// TwinCAT 3 PLC project lcls_plc_dream_vac
// ProgramVersion: 3.1.4022.7
// libraries:
//   LCLS General, * (SLAC)
//   LCLS Vacuum, * (SLAC - LCLS)
//   LCLSVacuumSerialDriverLib, * (SLAC - LCLS)
//   PMPS, * (SLAC - LCLS)
//   Tc2_SerialCom, * (Beckhoff Automation GmbH)
//   Tc2_Standard, * (Beckhoff Automation GmbH)
//   Tc2_System, * (Beckhoff Automation GmbH)
//   Tc2_Utilities, * (Beckhoff Automation GmbH)
//   Tc3_Module, * (Beckhoff Automation GmbH)
// project tree:
//   DUTs/ ST_TD400Control.TcDUT (not stored), ST_TD400Status.TcDUT (not stored)
//   GVLs/ GVL_FWM.TcGVL (not stored), GVL_PLC_Interface.TcGVL (not stored), GVL_Serial_Com.TcGVL (not stored), GVL_VAC_GAUGES.TcGVL (not stored), GVL_VAC_PUMPS.TcGVL (not stored), GVL_VAC_VALVES.TcGVL (not stored), GVL_Variables.TcGVL (not stored)
//   / PlcTask.TcTTO (not stored), Serial_COM.TcTTO (not stored)
//   POUs/Functions/ F_TurboIlkLogic.TcPOU (not stored)
//   POUs/ MAIN.TcPOU (not stored), PRG_COM.TcPOU (not stored), PRG_ECAT_CHECK.TcPOU (not stored), PRG_GAUGES.TcPOU (not stored), PRG_HV_ILK.TcPOU (not stored), PRG_COIL_PS_ILK.TcPOU (not stored), PRG_TURBO_PUMPS.TcPOU (not stored), PRG_VALVES.TcPOU (not stored)
//   POUs/TD400_Test/ FB_OERLIKON_TD400_COM.TcPOU, FB_OERLIKON_TD400_TO_PTM.TcPOU, FB_TD400SerialDriver.TcPOU (not stored), FB_TD400Transaction.TcPOU (not stored), F_CalcTD400Checksum.TcPOU (not stored)
//   POUs/TempFB_IE514/ FB_IE514.TcPOU (not stored)
// real-time tasks:
//   TASK PlcTask: cycle T#10ms, priority 20, ADS port 350
//   TASK Serial_COM: cycle T#2ms, priority 19, ADS port 351
// I/O:
//   DEVICE Device 1 (EtherCAT)
// variable links:
//   lcls_plc_dream_vac Instance <-> Device 1 (EtherCAT)/R20_DRL_03_CX0_EK1200/R20_DRL_03_E10_EL6001
//     Serial_COM Inputs/GVL_Serial_Com.stComIn_DREAM_DP3_PTM_01/D[0] <-> COM Inputs/Data In 0
//     Serial_COM Inputs/GVL_Serial_Com.stComIn_DREAM_DP3_PTM_01/D[10] <-> COM Inputs/Data In 10
//     Serial_COM Inputs/GVL_Serial_Com.stComIn_DREAM_DP3_PTM_01/D[11] <-> COM Inputs/Data In 11
//     Serial_COM Inputs/GVL_Serial_Com.stComIn_DREAM_DP3_PTM_01/D[12] <-> COM Inputs/Data In 12
//     Serial_COM Inputs/GVL_Serial_Com.stComIn_DREAM_DP3_PTM_01/D[13] <-> COM Inputs/Data In 13
//     Serial_COM Inputs/GVL_Serial_Com.stComIn_DREAM_DP3_PTM_01/D[14] <-> COM Inputs/Data In 14
//     Serial_COM Inputs/GVL_Serial_Com.stComIn_DREAM_DP3_PTM_01/D[15] <-> COM Inputs/Data In 15
//     Serial_COM Inputs/GVL_Serial_Com.stComIn_DREAM_DP3_PTM_01/D[16] <-> COM Inputs/Data In 16
//     Serial_COM Inputs/GVL_Serial_Com.stComIn_DREAM_DP3_PTM_01/D[17] <-> COM Inputs/Data In 17
//     Serial_COM Inputs/GVL_Serial_Com.stComIn_DREAM_DP3_PTM_01/D[18] <-> COM Inputs/Data In 18
//     Serial_COM Inputs/GVL_Serial_Com.stComIn_DREAM_DP3_PTM_01/D[19] <-> COM Inputs/Data In 19
//     Serial_COM Inputs/GVL_Serial_Com.stComIn_DREAM_DP3_PTM_01/D[1] <-> COM Inputs/Data In 1
//     Serial_COM Inputs/GVL_Serial_Com.stComIn_DREAM_DP3_PTM_01/D[20] <-> COM Inputs/Data In 20
//     Serial_COM Inputs/GVL_Serial_Com.stComIn_DREAM_DP3_PTM_01/D[21] <-> COM Inputs/Data In 21
//     Serial_COM Inputs/GVL_Serial_Com.stComIn_DREAM_DP3_PTM_01/D[2] <-> COM Inputs/Data In 2
//     Serial_COM Inputs/GVL_Serial_Com.stComIn_DREAM_DP3_PTM_01/D[3] <-> COM Inputs/Data In 3
//     Serial_COM Inputs/GVL_Serial_Com.stComIn_DREAM_DP3_PTM_01/D[4] <-> COM Inputs/Data In 4
//     Serial_COM Inputs/GVL_Serial_Com.stComIn_DREAM_DP3_PTM_01/D[5] <-> COM Inputs/Data In 5
//     Serial_COM Inputs/GVL_Serial_Com.stComIn_DREAM_DP3_PTM_01/D[6] <-> COM Inputs/Data In 6
//     Serial_COM Inputs/GVL_Serial_Com.stComIn_DREAM_DP3_PTM_01/D[7] <-> COM Inputs/Data In 7
//     Serial_COM Inputs/GVL_Serial_Com.stComIn_DREAM_DP3_PTM_01/D[8] <-> COM Inputs/Data In 8
//     Serial_COM Inputs/GVL_Serial_Com.stComIn_DREAM_DP3_PTM_01/D[9] <-> COM Inputs/Data In 9
//     Serial_COM Inputs/GVL_Serial_Com.stComIn_DREAM_DP3_PTM_01/Status <-> COM Inputs/Status
//     Serial_COM Outputs/GVL_Serial_Com.stComOut_DREAM_DP3_PTM_01/Ctrl <-> COM Outputs/Ctrl
//     Serial_COM Outputs/GVL_Serial_Com.stComOut_DREAM_DP3_PTM_01/D[0] <-> COM Outputs/Data Out 0
//     Serial_COM Outputs/GVL_Serial_Com.stComOut_DREAM_DP3_PTM_01/D[10] <-> COM Outputs/Data Out 10
//     Serial_COM Outputs/GVL_Serial_Com.stComOut_DREAM_DP3_PTM_01/D[11] <-> COM Outputs/Data Out 11
//     Serial_COM Outputs/GVL_Serial_Com.stComOut_DREAM_DP3_PTM_01/D[12] <-> COM Outputs/Data Out 12
//     Serial_COM Outputs/GVL_Serial_Com.stComOut_DREAM_DP3_PTM_01/D[13] <-> COM Outputs/Data Out 13
//     Serial_COM Outputs/GVL_Serial_Com.stComOut_DREAM_DP3_PTM_01/D[14] <-> COM Outputs/Data Out 14
//     Serial_COM Outputs/GVL_Serial_Com.stComOut_DREAM_DP3_PTM_01/D[15] <-> COM Outputs/Data Out 15
//     Serial_COM Outputs/GVL_Serial_Com.stComOut_DREAM_DP3_PTM_01/D[16] <-> COM Outputs/Data Out 16
//     Serial_COM Outputs/GVL_Serial_Com.stComOut_DREAM_DP3_PTM_01/D[17] <-> COM Outputs/Data Out 17
//     Serial_COM Outputs/GVL_Serial_Com.stComOut_DREAM_DP3_PTM_01/D[18] <-> COM Outputs/Data Out 18
//     Serial_COM Outputs/GVL_Serial_Com.stComOut_DREAM_DP3_PTM_01/D[19] <-> COM Outputs/Data Out 19
//     Serial_COM Outputs/GVL_Serial_Com.stComOut_DREAM_DP3_PTM_01/D[1] <-> COM Outputs/Data Out 1
//     Serial_COM Outputs/GVL_Serial_Com.stComOut_DREAM_DP3_PTM_01/D[20] <-> COM Outputs/Data Out 20
//     Serial_COM Outputs/GVL_Serial_Com.stComOut_DREAM_DP3_PTM_01/D[21] <-> COM Outputs/Data Out 21
//     Serial_COM Outputs/GVL_Serial_Com.stComOut_DREAM_DP3_PTM_01/D[2] <-> COM Outputs/Data Out 2
//     Serial_COM Outputs/GVL_Serial_Com.stComOut_DREAM_DP3_PTM_01/D[3] <-> COM Outputs/Data Out 3
//     Serial_COM Outputs/GVL_Serial_Com.stComOut_DREAM_DP3_PTM_01/D[4] <-> COM Outputs/Data Out 4
//     Serial_COM Outputs/GVL_Serial_Com.stComOut_DREAM_DP3_PTM_01/D[5] <-> COM Outputs/Data Out 5
//     Serial_COM Outputs/GVL_Serial_Com.stComOut_DREAM_DP3_PTM_01/D[6] <-> COM Outputs/Data Out 6
//     Serial_COM Outputs/GVL_Serial_Com.stComOut_DREAM_DP3_PTM_01/D[7] <-> COM Outputs/Data Out 7
//     Serial_COM Outputs/GVL_Serial_Com.stComOut_DREAM_DP3_PTM_01/D[8] <-> COM Outputs/Data Out 8
//     Serial_COM Outputs/GVL_Serial_Com.stComOut_DREAM_DP3_PTM_01/D[9] <-> COM Outputs/Data Out 9
//   lcls_plc_dream_vac Instance <-> Device 1 (EtherCAT)/R20_DRL_03_CX0_EK1200/R20_DRL_03_E11_EL6001
//     Serial_COM Inputs/GVL_Serial_Com.stComIn_DREAM_MC_PTM_01/D[0] <-> COM Inputs/Data In 0
//     Serial_COM Inputs/GVL_Serial_Com.stComIn_DREAM_MC_PTM_01/D[10] <-> COM Inputs/Data In 10
//     Serial_COM Inputs/GVL_Serial_Com.stComIn_DREAM_MC_PTM_01/D[11] <-> COM Inputs/Data In 11
//     Serial_COM Inputs/GVL_Serial_Com.stComIn_DREAM_MC_PTM_01/D[12] <-> COM Inputs/Data In 12
//     Serial_COM Inputs/GVL_Serial_Com.stComIn_DREAM_MC_PTM_01/D[13] <-> COM Inputs/Data In 13
//     Serial_COM Inputs/GVL_Serial_Com.stComIn_DREAM_MC_PTM_01/D[14] <-> COM Inputs/Data In 14
//     Serial_COM Inputs/GVL_Serial_Com.stComIn_DREAM_MC_PTM_01/D[15] <-> COM Inputs/Data In 15
//     Serial_COM Inputs/GVL_Serial_Com.stComIn_DREAM_MC_PTM_01/D[16] <-> COM Inputs/Data In 16
//     Serial_COM Inputs/GVL_Serial_Com.stComIn_DREAM_MC_PTM_01/D[17] <-> COM Inputs/Data In 17
//     Serial_COM Inputs/GVL_Serial_Com.stComIn_DREAM_MC_PTM_01/D[18] <-> COM Inputs/Data In 18
//     Serial_COM Inputs/GVL_Serial_Com.stComIn_DREAM_MC_PTM_01/D[19] <-> COM Inputs/Data In 19
//     Serial_COM Inputs/GVL_Serial_Com.stComIn_DREAM_MC_PTM_01/D[1] <-> COM Inputs/Data In 1
//     Serial_COM Inputs/GVL_Serial_Com.stComIn_DREAM_MC_PTM_01/D[20] <-> COM Inputs/Data In 20
//     Serial_COM Inputs/GVL_Serial_Com.stComIn_DREAM_MC_PTM_01/D[21] <-> COM Inputs/Data In 21
//     Serial_COM Inputs/GVL_Serial_Com.stComIn_DREAM_MC_PTM_01/D[2] <-> COM Inputs/Data In 2
//     Serial_COM Inputs/GVL_Serial_Com.stComIn_DREAM_MC_PTM_01/D[3] <-> COM Inputs/Data In 3
//     Serial_COM Inputs/GVL_Serial_Com.stComIn_DREAM_MC_PTM_01/D[4] <-> COM Inputs/Data In 4
//     Serial_COM Inputs/GVL_Serial_Com.stComIn_DREAM_MC_PTM_01/D[5] <-> COM Inputs/Data In 5
//     Serial_COM Inputs/GVL_Serial_Com.stComIn_DREAM_MC_PTM_01/D[6] <-> COM Inputs/Data In 6
//     Serial_COM Inputs/GVL_Serial_Com.stComIn_DREAM_MC_PTM_01/D[7] <-> COM Inputs/Data In 7
//     Serial_COM Inputs/GVL_Serial_Com.stComIn_DREAM_MC_PTM_01/D[8] <-> COM Inputs/Data In 8
//     Serial_COM Inputs/GVL_Serial_Com.stComIn_DREAM_MC_PTM_01/D[9] <-> COM Inputs/Data In 9
//     Serial_COM Inputs/GVL_Serial_Com.stComIn_DREAM_MC_PTM_01/Status <-> COM Inputs/Status
//     Serial_COM Outputs/GVL_Serial_Com.stComOut_DREAM_MC_PTM_01/Ctrl <-> COM Outputs/Ctrl
//     Serial_COM Outputs/GVL_Serial_Com.stComOut_DREAM_MC_PTM_01/D[0] <-> COM Outputs/Data Out 0
//     Serial_COM Outputs/GVL_Serial_Com.stComOut_DREAM_MC_PTM_01/D[10] <-> COM Outputs/Data Out 10
//     Serial_COM Outputs/GVL_Serial_Com.stComOut_DREAM_MC_PTM_01/D[11] <-> COM Outputs/Data Out 11
//     Serial_COM Outputs/GVL_Serial_Com.stComOut_DREAM_MC_PTM_01/D[12] <-> COM Outputs/Data Out 12
//     Serial_COM Outputs/GVL_Serial_Com.stComOut_DREAM_MC_PTM_01/D[13] <-> COM Outputs/Data Out 13
//     Serial_COM Outputs/GVL_Serial_Com.stComOut_DREAM_MC_PTM_01/D[14] <-> COM Outputs/Data Out 14
//     Serial_COM Outputs/GVL_Serial_Com.stComOut_DREAM_MC_PTM_01/D[15] <-> COM Outputs/Data Out 15
//     Serial_COM Outputs/GVL_Serial_Com.stComOut_DREAM_MC_PTM_01/D[16] <-> COM Outputs/Data Out 16
//     Serial_COM Outputs/GVL_Serial_Com.stComOut_DREAM_MC_PTM_01/D[17] <-> COM Outputs/Data Out 17
//     Serial_COM Outputs/GVL_Serial_Com.stComOut_DREAM_MC_PTM_01/D[18] <-> COM Outputs/Data Out 18
//     Serial_COM Outputs/GVL_Serial_Com.stComOut_DREAM_MC_PTM_01/D[19] <-> COM Outputs/Data Out 19
//     Serial_COM Outputs/GVL_Serial_Com.stComOut_DREAM_MC_PTM_01/D[1] <-> COM Outputs/Data Out 1
//     Serial_COM Outputs/GVL_Serial_Com.stComOut_DREAM_MC_PTM_01/D[20] <-> COM Outputs/Data Out 20
//     Serial_COM Outputs/GVL_Serial_Com.stComOut_DREAM_MC_PTM_01/D[21] <-> COM Outputs/Data Out 21
//     Serial_COM Outputs/GVL_Serial_Com.stComOut_DREAM_MC_PTM_01/D[2] <-> COM Outputs/Data Out 2
//     Serial_COM Outputs/GVL_Serial_Com.stComOut_DREAM_MC_PTM_01/D[3] <-> COM Outputs/Data Out 3
//     Serial_COM Outputs/GVL_Serial_Com.stComOut_DREAM_MC_PTM_01/D[4] <-> COM Outputs/Data Out 4
//     Serial_COM Outputs/GVL_Serial_Com.stComOut_DREAM_MC_PTM_01/D[5] <-> COM Outputs/Data Out 5
//     Serial_COM Outputs/GVL_Serial_Com.stComOut_DREAM_MC_PTM_01/D[6] <-> COM Outputs/Data Out 6
//     Serial_COM Outputs/GVL_Serial_Com.stComOut_DREAM_MC_PTM_01/D[7] <-> COM Outputs/Data Out 7
//     Serial_COM Outputs/GVL_Serial_Com.stComOut_DREAM_MC_PTM_01/D[8] <-> COM Outputs/Data Out 8
//     Serial_COM Outputs/GVL_Serial_Com.stComOut_DREAM_MC_PTM_01/D[9] <-> COM Outputs/Data Out 9
//   lcls_plc_dream_vac Instance <-> Device 1 (EtherCAT)/R20_DRL_03_CX0_EK1200/R20_DRL_03_E12_EL6001
//     Serial_COM Inputs/GVL_Serial_Com.stComIn_DREAM_MC_PTM_02/D[0] <-> COM Inputs/Data In 0
//     Serial_COM Inputs/GVL_Serial_Com.stComIn_DREAM_MC_PTM_02/D[10] <-> COM Inputs/Data In 10
//     Serial_COM Inputs/GVL_Serial_Com.stComIn_DREAM_MC_PTM_02/D[11] <-> COM Inputs/Data In 11
//     Serial_COM Inputs/GVL_Serial_Com.stComIn_DREAM_MC_PTM_02/D[12] <-> COM Inputs/Data In 12
//     Serial_COM Inputs/GVL_Serial_Com.stComIn_DREAM_MC_PTM_02/D[13] <-> COM Inputs/Data In 13
//     Serial_COM Inputs/GVL_Serial_Com.stComIn_DREAM_MC_PTM_02/D[14] <-> COM Inputs/Data In 14
//     Serial_COM Inputs/GVL_Serial_Com.stComIn_DREAM_MC_PTM_02/D[15] <-> COM Inputs/Data In 15
//     Serial_COM Inputs/GVL_Serial_Com.stComIn_DREAM_MC_PTM_02/D[16] <-> COM Inputs/Data In 16
//     Serial_COM Inputs/GVL_Serial_Com.stComIn_DREAM_MC_PTM_02/D[17] <-> COM Inputs/Data In 17
//     Serial_COM Inputs/GVL_Serial_Com.stComIn_DREAM_MC_PTM_02/D[18] <-> COM Inputs/Data In 18
//     Serial_COM Inputs/GVL_Serial_Com.stComIn_DREAM_MC_PTM_02/D[19] <-> COM Inputs/Data In 19
//     Serial_COM Inputs/GVL_Serial_Com.stComIn_DREAM_MC_PTM_02/D[1] <-> COM Inputs/Data In 1
//     Serial_COM Inputs/GVL_Serial_Com.stComIn_DREAM_MC_PTM_02/D[20] <-> COM Inputs/Data In 20
//     Serial_COM Inputs/GVL_Serial_Com.stComIn_DREAM_MC_PTM_02/D[21] <-> COM Inputs/Data In 21
//     Serial_COM Inputs/GVL_Serial_Com.stComIn_DREAM_MC_PTM_02/D[2] <-> COM Inputs/Data In 2
//     Serial_COM Inputs/GVL_Serial_Com.stComIn_DREAM_MC_PTM_02/D[3] <-> COM Inputs/Data In 3
//     Serial_COM Inputs/GVL_Serial_Com.stComIn_DREAM_MC_PTM_02/D[4] <-> COM Inputs/Data In 4
//     Serial_COM Inputs/GVL_Serial_Com.stComIn_DREAM_MC_PTM_02/D[5] <-> COM Inputs/Data In 5
//     Serial_COM Inputs/GVL_Serial_Com.stComIn_DREAM_MC_PTM_02/D[6] <-> COM Inputs/Data In 6
//     Serial_COM Inputs/GVL_Serial_Com.stComIn_DREAM_MC_PTM_02/D[7] <-> COM Inputs/Data In 7
//     Serial_COM Inputs/GVL_Serial_Com.stComIn_DREAM_MC_PTM_02/D[8] <-> COM Inputs/Data In 8
//     Serial_COM Inputs/GVL_Serial_Com.stComIn_DREAM_MC_PTM_02/D[9] <-> COM Inputs/Data In 9
//     Serial_COM Inputs/GVL_Serial_Com.stComIn_DREAM_MC_PTM_02/Status <-> COM Inputs/Status
//     Serial_COM Outputs/GVL_Serial_Com.stComOut_DREAM_MC_PTM_02/Ctrl <-> COM Outputs/Ctrl
//     Serial_COM Outputs/GVL_Serial_Com.stComOut_DREAM_MC_PTM_02/D[0] <-> COM Outputs/Data Out 0
//     Serial_COM Outputs/GVL_Serial_Com.stComOut_DREAM_MC_PTM_02/D[10] <-> COM Outputs/Data Out 10
//     Serial_COM Outputs/GVL_Serial_Com.stComOut_DREAM_MC_PTM_02/D[11] <-> COM Outputs/Data Out 11
//     Serial_COM Outputs/GVL_Serial_Com.stComOut_DREAM_MC_PTM_02/D[12] <-> COM Outputs/Data Out 12
//     Serial_COM Outputs/GVL_Serial_Com.stComOut_DREAM_MC_PTM_02/D[13] <-> COM Outputs/Data Out 13
//     Serial_COM Outputs/GVL_Serial_Com.stComOut_DREAM_MC_PTM_02/D[14] <-> COM Outputs/Data Out 14
//     Serial_COM Outputs/GVL_Serial_Com.stComOut_DREAM_MC_PTM_02/D[15] <-> COM Outputs/Data Out 15
//     Serial_COM Outputs/GVL_Serial_Com.stComOut_DREAM_MC_PTM_02/D[16] <-> COM Outputs/Data Out 16
//     Serial_COM Outputs/GVL_Serial_Com.stComOut_DREAM_MC_PTM_02/D[17] <-> COM Outputs/Data Out 17
//     Serial_COM Outputs/GVL_Serial_Com.stComOut_DREAM_MC_PTM_02/D[18] <-> COM Outputs/Data Out 18
//     Serial_COM Outputs/GVL_Serial_Com.stComOut_DREAM_MC_PTM_02/D[19] <-> COM Outputs/Data Out 19
//     Serial_COM Outputs/GVL_Serial_Com.stComOut_DREAM_MC_PTM_02/D[1] <-> COM Outputs/Data Out 1
//     Serial_COM Outputs/GVL_Serial_Com.stComOut_DREAM_MC_PTM_02/D[20] <-> COM Outputs/Data Out 20
//     Serial_COM Outputs/GVL_Serial_Com.stComOut_DREAM_MC_PTM_02/D[21] <-> COM Outputs/Data Out 21
//     Serial_COM Outputs/GVL_Serial_Com.stComOut_DREAM_MC_PTM_02/D[2] <-> COM Outputs/Data Out 2
//     Serial_COM Outputs/GVL_Serial_Com.stComOut_DREAM_MC_PTM_02/D[3] <-> COM Outputs/Data Out 3
//     Serial_COM Outputs/GVL_Serial_Com.stComOut_DREAM_MC_PTM_02/D[4] <-> COM Outputs/Data Out 4
//     Serial_COM Outputs/GVL_Serial_Com.stComOut_DREAM_MC_PTM_02/D[5] <-> COM Outputs/Data Out 5
//     Serial_COM Outputs/GVL_Serial_Com.stComOut_DREAM_MC_PTM_02/D[6] <-> COM Outputs/Data Out 6
//     Serial_COM Outputs/GVL_Serial_Com.stComOut_DREAM_MC_PTM_02/D[7] <-> COM Outputs/Data Out 7
//     Serial_COM Outputs/GVL_Serial_Com.stComOut_DREAM_MC_PTM_02/D[8] <-> COM Outputs/Data Out 8
//     Serial_COM Outputs/GVL_Serial_Com.stComOut_DREAM_MC_PTM_02/D[9] <-> COM Outputs/Data Out 9
//   lcls_plc_dream_vac Instance <-> Device 1 (EtherCAT)/R20_DRL_03_CX0_EK1200/R20_DRL_03_E14_EL6695
//     PlcTask Inputs/GVL_PLC_Interface.bEcatBridge_External_device_not_connected <-> SYNC Inputs/External device not connected
//     PlcTask Inputs/GVL_PLC_Interface.bEcatBridge_TxPDO_state <-> SYNC Inputs/TxPDO state
//     PlcTask Inputs/GVL_PLC_Interface.bEcatBridge_WcState <-> WcState/WcStateIn
//     PlcTask Inputs/GVL_PLC_Interface.sHUTCH_PLC_NAME <-> IO Inputs/HUTCH_PLC_NAME
//     PlcTask Outputs/GVL_PLC_Interface.bDREAM_HV_SAFETY_ENABLE <-> IO Outputs/DREAM_HV_SAFETY_ENABLE
//     PlcTask Outputs/GVL_PLC_Interface.bDREAM_MAIN_xAT_VAC <-> IO Outputs/DREAM_MAIN_xAT_VAC
//     PlcTask Outputs/GVL_PLC_Interface.bDREAM_MAIN_xPRESS_OK <-> IO Outputs/DREAM_MAIN_xPRESS_OK
//     PlcTask Outputs/GVL_PLC_Interface.bDREAM_TURBOS_ALL_AtSpd <-> IO Outputs/DREAM_TURBOS_ALL_AtSpd
//     PlcTask Outputs/GVL_PLC_Interface.fDREAM_MAIN_rPRESS <-> IO Outputs/DREAM_MAIN_rPRESS
//     PlcTask Outputs/GVL_PLC_Interface.sENDSTATION_PLC_NAME <-> IO Outputs/ENDSTATION_PLC_NAME
//   lcls_plc_dream_vac Instance <-> Device 1 (EtherCAT)/R20_DRL_03_CX0_EK1200/R20_DRL_03_E15_EL1122/K4S8_DRL_03_EK0_EK1100/K4S8_DRL_03_E10_EL1004
//     PlcTask Inputs/GVL_VAC_VALVES.DREAM_DP1_VRC_01.i_xClsLS <-> Channel 2/Input
//     PlcTask Inputs/GVL_VAC_VALVES.DREAM_DP1_VRC_02.i_xClsLS <-> Channel 4/Input
//     PlcTask Inputs/GVL_VAC_VALVES.DREAM_DP1_VRC_01.i_xOpnLS <-> Channel 1/Input
//     PlcTask Inputs/GVL_VAC_VALVES.DREAM_DP1_VRC_02.i_xOpnLS <-> Channel 3/Input
//   lcls_plc_dream_vac Instance <-> Device 1 (EtherCAT)/R20_DRL_03_CX0_EK1200/R20_DRL_03_E15_EL1122/K4S8_DRL_03_EK0_EK1100/K4S8_DRL_03_E11_EL2004
//     PlcTask Outputs/GVL_VAC_VALVES.DREAM_DP1_VRC_01.q_xOPN_DO <-> Channel 2/Output
//     PlcTask Outputs/GVL_VAC_VALVES.DREAM_DP1_VRC_02.q_xCLS_DO <-> Channel 1/Output
//   lcls_plc_dream_vac Instance <-> Device 1 (EtherCAT)/R20_DRL_03_CX0_EK1200/R20_DRL_03_E15_EL1122/K4S8_DRL_03_EK0_EK1100/K4S8_DRL_03_E12_EL6021
//     Serial_COM Inputs/GVL_Serial_Com.stComIn_DREAM_NC_PTM_01/D[0] <-> COM TxPDO-Map Inputs/Data In 0
//     Serial_COM Inputs/GVL_Serial_Com.stComIn_DREAM_NC_PTM_01/D[10] <-> COM TxPDO-Map Inputs/Data In 10
//     Serial_COM Inputs/GVL_Serial_Com.stComIn_DREAM_NC_PTM_01/D[11] <-> COM TxPDO-Map Inputs/Data In 11
//     Serial_COM Inputs/GVL_Serial_Com.stComIn_DREAM_NC_PTM_01/D[12] <-> COM TxPDO-Map Inputs/Data In 12
//     Serial_COM Inputs/GVL_Serial_Com.stComIn_DREAM_NC_PTM_01/D[13] <-> COM TxPDO-Map Inputs/Data In 13
//     Serial_COM Inputs/GVL_Serial_Com.stComIn_DREAM_NC_PTM_01/D[14] <-> COM TxPDO-Map Inputs/Data In 14
//     Serial_COM Inputs/GVL_Serial_Com.stComIn_DREAM_NC_PTM_01/D[15] <-> COM TxPDO-Map Inputs/Data In 15
//     Serial_COM Inputs/GVL_Serial_Com.stComIn_DREAM_NC_PTM_01/D[16] <-> COM TxPDO-Map Inputs/Data In 16
//     Serial_COM Inputs/GVL_Serial_Com.stComIn_DREAM_NC_PTM_01/D[17] <-> COM TxPDO-Map Inputs/Data In 17
//     Serial_COM Inputs/GVL_Serial_Com.stComIn_DREAM_NC_PTM_01/D[18] <-> COM TxPDO-Map Inputs/Data In 18
//     Serial_COM Inputs/GVL_Serial_Com.stComIn_DREAM_NC_PTM_01/D[19] <-> COM TxPDO-Map Inputs/Data In 19
//     Serial_COM Inputs/GVL_Serial_Com.stComIn_DREAM_NC_PTM_01/D[1] <-> COM TxPDO-Map Inputs/Data In 1
//     Serial_COM Inputs/GVL_Serial_Com.stComIn_DREAM_NC_PTM_01/D[20] <-> COM TxPDO-Map Inputs/Data In 20
//     Serial_COM Inputs/GVL_Serial_Com.stComIn_DREAM_NC_PTM_01/D[21] <-> COM TxPDO-Map Inputs/Data In 21
//     Serial_COM Inputs/GVL_Serial_Com.stComIn_DREAM_NC_PTM_01/D[2] <-> COM TxPDO-Map Inputs/Data In 2
//     Serial_COM Inputs/GVL_Serial_Com.stComIn_DREAM_NC_PTM_01/D[3] <-> COM TxPDO-Map Inputs/Data In 3
//     Serial_COM Inputs/GVL_Serial_Com.stComIn_DREAM_NC_PTM_01/D[4] <-> COM TxPDO-Map Inputs/Data In 4
//     Serial_COM Inputs/GVL_Serial_Com.stComIn_DREAM_NC_PTM_01/D[5] <-> COM TxPDO-Map Inputs/Data In 5
//     Serial_COM Inputs/GVL_Serial_Com.stComIn_DREAM_NC_PTM_01/D[6] <-> COM TxPDO-Map Inputs/Data In 6
//     Serial_COM Inputs/GVL_Serial_Com.stComIn_DREAM_NC_PTM_01/D[7] <-> COM TxPDO-Map Inputs/Data In 7
//     Serial_COM Inputs/GVL_Serial_Com.stComIn_DREAM_NC_PTM_01/D[8] <-> COM TxPDO-Map Inputs/Data In 8
//     Serial_COM Inputs/GVL_Serial_Com.stComIn_DREAM_NC_PTM_01/D[9] <-> COM TxPDO-Map Inputs/Data In 9
//     Serial_COM Inputs/GVL_Serial_Com.stComIn_DREAM_NC_PTM_01/Status <-> COM TxPDO-Map Inputs/Status
//     Serial_COM Outputs/GVL_Serial_Com.stComOut_DREAM_NC_PTM_01/Ctrl <-> COM RxPDO-Map Outputs/Ctrl
//     Serial_COM Outputs/GVL_Serial_Com.stComOut_DREAM_NC_PTM_01/D[0] <-> COM RxPDO-Map Outputs/Data Out 0
//     Serial_COM Outputs/GVL_Serial_Com.stComOut_DREAM_NC_PTM_01/D[10] <-> COM RxPDO-Map Outputs/Data Out 10
//     Serial_COM Outputs/GVL_Serial_Com.stComOut_DREAM_NC_PTM_01/D[11] <-> COM RxPDO-Map Outputs/Data Out 11
//     Serial_COM Outputs/GVL_Serial_Com.stComOut_DREAM_NC_PTM_01/D[12] <-> COM RxPDO-Map Outputs/Data Out 12
//     Serial_COM Outputs/GVL_Serial_Com.stComOut_DREAM_NC_PTM_01/D[13] <-> COM RxPDO-Map Outputs/Data Out 13
//     Serial_COM Outputs/GVL_Serial_Com.stComOut_DREAM_NC_PTM_01/D[14] <-> COM RxPDO-Map Outputs/Data Out 14
//     Serial_COM Outputs/GVL_Serial_Com.stComOut_DREAM_NC_PTM_01/D[15] <-> COM RxPDO-Map Outputs/Data Out 15
//     Serial_COM Outputs/GVL_Serial_Com.stComOut_DREAM_NC_PTM_01/D[16] <-> COM RxPDO-Map Outputs/Data Out 16
//     Serial_COM Outputs/GVL_Serial_Com.stComOut_DREAM_NC_PTM_01/D[17] <-> COM RxPDO-Map Outputs/Data Out 17
//     Serial_COM Outputs/GVL_Serial_Com.stComOut_DREAM_NC_PTM_01/D[18] <-> COM RxPDO-Map Outputs/Data Out 18
//     Serial_COM Outputs/GVL_Serial_Com.stComOut_DREAM_NC_PTM_01/D[19] <-> COM RxPDO-Map Outputs/Data Out 19
//     Serial_COM Outputs/GVL_Serial_Com.stComOut_DREAM_NC_PTM_01/D[1] <-> COM RxPDO-Map Outputs/Data Out 1
//     Serial_COM Outputs/GVL_Serial_Com.stComOut_DREAM_NC_PTM_01/D[20] <-> COM RxPDO-Map Outputs/Data Out 20
//     Serial_COM Outputs/GVL_Serial_Com.stComOut_DREAM_NC_PTM_01/D[21] <-> COM RxPDO-Map Outputs/Data Out 21
//     Serial_COM Outputs/GVL_Serial_Com.stComOut_DREAM_NC_PTM_01/D[2] <-> COM RxPDO-Map Outputs/Data Out 2
//     Serial_COM Outputs/GVL_Serial_Com.stComOut_DREAM_NC_PTM_01/D[3] <-> COM RxPDO-Map Outputs/Data Out 3
//     Serial_COM Outputs/GVL_Serial_Com.stComOut_DREAM_NC_PTM_01/D[4] <-> COM RxPDO-Map Outputs/Data Out 4
//     Serial_COM Outputs/GVL_Serial_Com.stComOut_DREAM_NC_PTM_01/D[5] <-> COM RxPDO-Map Outputs/Data Out 5
//     Serial_COM Outputs/GVL_Serial_Com.stComOut_DREAM_NC_PTM_01/D[6] <-> COM RxPDO-Map Outputs/Data Out 6
//     Serial_COM Outputs/GVL_Serial_Com.stComOut_DREAM_NC_PTM_01/D[7] <-> COM RxPDO-Map Outputs/Data Out 7
//     Serial_COM Outputs/GVL_Serial_Com.stComOut_DREAM_NC_PTM_01/D[8] <-> COM RxPDO-Map Outputs/Data Out 8
//     Serial_COM Outputs/GVL_Serial_Com.stComOut_DREAM_NC_PTM_01/D[9] <-> COM RxPDO-Map Outputs/Data Out 9
//   lcls_plc_dream_vac Instance <-> Device 1 (EtherCAT)/R20_DRL_03_CX0_EK1200/R20_DRL_03_E15_EL1122/K4S8_DRL_03_EK0_EK1100/K4S8_DRL_03_E13_EL1004
//     PlcTask Inputs/GVL_VAC_PUMPS.DREAM_NC_PTM_01.i_xAtSpd <-> Channel 1/Input
//     PlcTask Inputs/GVL_VAC_PUMPS.DREAM_NC_PTM_01.i_xFaultNC <-> Channel 3/Input
//     PlcTask Inputs/GVL_VAC_PUMPS.DREAM_NC_PTM_01.i_xRemote <-> Channel 2/Input
//   lcls_plc_dream_vac Instance <-> Device 1 (EtherCAT)/R20_DRL_03_CX0_EK1200/R20_DRL_03_E15_EL1122/K4S8_DRL_03_EK0_EK1100/K4S8_DRL_03_E14_EL2004
//     PlcTask Outputs/GVL_VAC_PUMPS.DREAM_NC_PTM_01.q_PumpingStation <-> Channel 3/Output
//     PlcTask Outputs/GVL_VAC_PUMPS.DREAM_NC_PTM_01.q_RunDO <-> Channel 1/Output
//     PlcTask Outputs/GVL_VAC_PUMPS.DREAM_NC_PTM_01.q_xRemote <-> Channel 2/Output
//   lcls_plc_dream_vac Instance <-> Device 1 (EtherCAT)/R20_DRL_03_CX0_EK1200/R20_DRL_03_E15_EL1122/K4S8_DRL_03_EK0_EK1100/K4S8_DRL_03_E15_EL6021
//     Serial_COM Inputs/GVL_Serial_Com.stComIn_DREAM_NC_PTM_02/D[0] <-> COM TxPDO-Map Inputs/Data In 0
//     Serial_COM Inputs/GVL_Serial_Com.stComIn_DREAM_NC_PTM_02/D[10] <-> COM TxPDO-Map Inputs/Data In 10
//     Serial_COM Inputs/GVL_Serial_Com.stComIn_DREAM_NC_PTM_02/D[11] <-> COM TxPDO-Map Inputs/Data In 11
//     Serial_COM Inputs/GVL_Serial_Com.stComIn_DREAM_NC_PTM_02/D[12] <-> COM TxPDO-Map Inputs/Data In 12
//     Serial_COM Inputs/GVL_Serial_Com.stComIn_DREAM_NC_PTM_02/D[13] <-> COM TxPDO-Map Inputs/Data In 13
//     Serial_COM Inputs/GVL_Serial_Com.stComIn_DREAM_NC_PTM_02/D[14] <-> COM TxPDO-Map Inputs/Data In 14
//     Serial_COM Inputs/GVL_Serial_Com.stComIn_DREAM_NC_PTM_02/D[15] <-> COM TxPDO-Map Inputs/Data In 15
//     Serial_COM Inputs/GVL_Serial_Com.stComIn_DREAM_NC_PTM_02/D[16] <-> COM TxPDO-Map Inputs/Data In 16
//     Serial_COM Inputs/GVL_Serial_Com.stComIn_DREAM_NC_PTM_02/D[17] <-> COM TxPDO-Map Inputs/Data In 17
//     Serial_COM Inputs/GVL_Serial_Com.stComIn_DREAM_NC_PTM_02/D[18] <-> COM TxPDO-Map Inputs/Data In 18
//     Serial_COM Inputs/GVL_Serial_Com.stComIn_DREAM_NC_PTM_02/D[19] <-> COM TxPDO-Map Inputs/Data In 19
//     Serial_COM Inputs/GVL_Serial_Com.stComIn_DREAM_NC_PTM_02/D[1] <-> COM TxPDO-Map Inputs/Data In 1
//     Serial_COM Inputs/GVL_Serial_Com.stComIn_DREAM_NC_PTM_02/D[20] <-> COM TxPDO-Map Inputs/Data In 20
//     Serial_COM Inputs/GVL_Serial_Com.stComIn_DREAM_NC_PTM_02/D[21] <-> COM TxPDO-Map Inputs/Data In 21
//     Serial_COM Inputs/GVL_Serial_Com.stComIn_DREAM_NC_PTM_02/D[2] <-> COM TxPDO-Map Inputs/Data In 2
//     Serial_COM Inputs/GVL_Serial_Com.stComIn_DREAM_NC_PTM_02/D[3] <-> COM TxPDO-Map Inputs/Data In 3
//     Serial_COM Inputs/GVL_Serial_Com.stComIn_DREAM_NC_PTM_02/D[4] <-> COM TxPDO-Map Inputs/Data In 4
//     Serial_COM Inputs/GVL_Serial_Com.stComIn_DREAM_NC_PTM_02/D[5] <-> COM TxPDO-Map Inputs/Data In 5
//     Serial_COM Inputs/GVL_Serial_Com.stComIn_DREAM_NC_PTM_02/D[6] <-> COM TxPDO-Map Inputs/Data In 6
//     Serial_COM Inputs/GVL_Serial_Com.stComIn_DREAM_NC_PTM_02/D[7] <-> COM TxPDO-Map Inputs/Data In 7
//     Serial_COM Inputs/GVL_Serial_Com.stComIn_DREAM_NC_PTM_02/D[8] <-> COM TxPDO-Map Inputs/Data In 8
//     Serial_COM Inputs/GVL_Serial_Com.stComIn_DREAM_NC_PTM_02/D[9] <-> COM TxPDO-Map Inputs/Data In 9
//     Serial_COM Inputs/GVL_Serial_Com.stComIn_DREAM_NC_PTM_02/Status <-> COM TxPDO-Map Inputs/Status
//     Serial_COM Outputs/GVL_Serial_Com.stComOut_DREAM_NC_PTM_02/Ctrl <-> COM RxPDO-Map Outputs/Ctrl
//     Serial_COM Outputs/GVL_Serial_Com.stComOut_DREAM_NC_PTM_02/D[0] <-> COM RxPDO-Map Outputs/Data Out 0
//     Serial_COM Outputs/GVL_Serial_Com.stComOut_DREAM_NC_PTM_02/D[10] <-> COM RxPDO-Map Outputs/Data Out 10
//     Serial_COM Outputs/GVL_Serial_Com.stComOut_DREAM_NC_PTM_02/D[11] <-> COM RxPDO-Map Outputs/Data Out 11
//     Serial_COM Outputs/GVL_Serial_Com.stComOut_DREAM_NC_PTM_02/D[12] <-> COM RxPDO-Map Outputs/Data Out 12
//     Serial_COM Outputs/GVL_Serial_Com.stComOut_DREAM_NC_PTM_02/D[13] <-> COM RxPDO-Map Outputs/Data Out 13
//     Serial_COM Outputs/GVL_Serial_Com.stComOut_DREAM_NC_PTM_02/D[14] <-> COM RxPDO-Map Outputs/Data Out 14
//     Serial_COM Outputs/GVL_Serial_Com.stComOut_DREAM_NC_PTM_02/D[15] <-> COM RxPDO-Map Outputs/Data Out 15
//     Serial_COM Outputs/GVL_Serial_Com.stComOut_DREAM_NC_PTM_02/D[16] <-> COM RxPDO-Map Outputs/Data Out 16
//     Serial_COM Outputs/GVL_Serial_Com.stComOut_DREAM_NC_PTM_02/D[17] <-> COM RxPDO-Map Outputs/Data Out 17
//     Serial_COM Outputs/GVL_Serial_Com.stComOut_DREAM_NC_PTM_02/D[18] <-> COM RxPDO-Map Outputs/Data Out 18
//     Serial_COM Outputs/GVL_Serial_Com.stComOut_DREAM_NC_PTM_02/D[19] <-> COM RxPDO-Map Outputs/Data Out 19
//     Serial_COM Outputs/GVL_Serial_Com.stComOut_DREAM_NC_PTM_02/D[1] <-> COM RxPDO-Map Outputs/Data Out 1
//     Serial_COM Outputs/GVL_Serial_Com.stComOut_DREAM_NC_PTM_02/D[20] <-> COM RxPDO-Map Outputs/Data Out 20
//     Serial_COM Outputs/GVL_Serial_Com.stComOut_DREAM_NC_PTM_02/D[21] <-> COM RxPDO-Map Outputs/Data Out 21
//     Serial_COM Outputs/GVL_Serial_Com.stComOut_DREAM_NC_PTM_02/D[2] <-> COM RxPDO-Map Outputs/Data Out 2
//     Serial_COM Outputs/GVL_Serial_Com.stComOut_DREAM_NC_PTM_02/D[3] <-> COM RxPDO-Map Outputs/Data Out 3
//     Serial_COM Outputs/GVL_Serial_Com.stComOut_DREAM_NC_PTM_02/D[4] <-> COM RxPDO-Map Outputs/Data Out 4
//     Serial_COM Outputs/GVL_Serial_Com.stComOut_DREAM_NC_PTM_02/D[5] <-> COM RxPDO-Map Outputs/Data Out 5
//     Serial_COM Outputs/GVL_Serial_Com.stComOut_DREAM_NC_PTM_02/D[6] <-> COM RxPDO-Map Outputs/Data Out 6
//     Serial_COM Outputs/GVL_Serial_Com.stComOut_DREAM_NC_PTM_02/D[7] <-> COM RxPDO-Map Outputs/Data Out 7
//     Serial_COM Outputs/GVL_Serial_Com.stComOut_DREAM_NC_PTM_02/D[8] <-> COM RxPDO-Map Outputs/Data Out 8
//     Serial_COM Outputs/GVL_Serial_Com.stComOut_DREAM_NC_PTM_02/D[9] <-> COM RxPDO-Map Outputs/Data Out 9
//   lcls_plc_dream_vac Instance <-> Device 1 (EtherCAT)/R20_DRL_03_CX0_EK1200/R20_DRL_03_E15_EL1122/K4S8_DRL_03_EK0_EK1100/K4S8_DRL_03_E16_EL1004
//     PlcTask Inputs/GVL_VAC_PUMPS.DREAM_NC_PTM_02.i_xAtSpd <-> Channel 1/Input
//     PlcTask Inputs/GVL_VAC_PUMPS.DREAM_NC_PTM_02.i_xFaultNC <-> Channel 3/Input
//     PlcTask Inputs/GVL_VAC_PUMPS.DREAM_NC_PTM_02.i_xRemote <-> Channel 2/Input
//   lcls_plc_dream_vac Instance <-> Device 1 (EtherCAT)/R20_DRL_03_CX0_EK1200/R20_DRL_03_E15_EL1122/K4S8_DRL_03_EK0_EK1100/K4S8_DRL_03_E17_EL2004
//     PlcTask Outputs/GVL_VAC_PUMPS.DREAM_NC_PTM_02.q_PumpingStation <-> Channel 3/Output
//     PlcTask Outputs/GVL_VAC_PUMPS.DREAM_NC_PTM_02.q_RunDO <-> Channel 1/Output
//     PlcTask Outputs/GVL_VAC_PUMPS.DREAM_NC_PTM_02.q_xRemote <-> Channel 2/Output
//   lcls_plc_dream_vac Instance <-> Device 1 (EtherCAT)/R20_DRL_03_CX0_EK1200/R20_DRL_03_E15_EL1122/K4S8_DRL_03_EK0_EK1100/K4S8_DRL_03_E18_EL6021
//     Serial_COM Inputs/GVL_Serial_Com.stComIn_DREAM_DP1_PTM_01/D[0] <-> COM TxPDO-Map Inputs/Data In 0
//     Serial_COM Inputs/GVL_Serial_Com.stComIn_DREAM_DP1_PTM_01/D[10] <-> COM TxPDO-Map Inputs/Data In 10
//     Serial_COM Inputs/GVL_Serial_Com.stComIn_DREAM_DP1_PTM_01/D[11] <-> COM TxPDO-Map Inputs/Data In 11
//     Serial_COM Inputs/GVL_Serial_Com.stComIn_DREAM_DP1_PTM_01/D[12] <-> COM TxPDO-Map Inputs/Data In 12
//     Serial_COM Inputs/GVL_Serial_Com.stComIn_DREAM_DP1_PTM_01/D[13] <-> COM TxPDO-Map Inputs/Data In 13
//     Serial_COM Inputs/GVL_Serial_Com.stComIn_DREAM_DP1_PTM_01/D[14] <-> COM TxPDO-Map Inputs/Data In 14
//     Serial_COM Inputs/GVL_Serial_Com.stComIn_DREAM_DP1_PTM_01/D[15] <-> COM TxPDO-Map Inputs/Data In 15
//     Serial_COM Inputs/GVL_Serial_Com.stComIn_DREAM_DP1_PTM_01/D[16] <-> COM TxPDO-Map Inputs/Data In 16
//     Serial_COM Inputs/GVL_Serial_Com.stComIn_DREAM_DP1_PTM_01/D[17] <-> COM TxPDO-Map Inputs/Data In 17
//     Serial_COM Inputs/GVL_Serial_Com.stComIn_DREAM_DP1_PTM_01/D[18] <-> COM TxPDO-Map Inputs/Data In 18
//     Serial_COM Inputs/GVL_Serial_Com.stComIn_DREAM_DP1_PTM_01/D[19] <-> COM TxPDO-Map Inputs/Data In 19
//     Serial_COM Inputs/GVL_Serial_Com.stComIn_DREAM_DP1_PTM_01/D[1] <-> COM TxPDO-Map Inputs/Data In 1
//     Serial_COM Inputs/GVL_Serial_Com.stComIn_DREAM_DP1_PTM_01/D[20] <-> COM TxPDO-Map Inputs/Data In 20
//     Serial_COM Inputs/GVL_Serial_Com.stComIn_DREAM_DP1_PTM_01/D[21] <-> COM TxPDO-Map Inputs/Data In 21
//     Serial_COM Inputs/GVL_Serial_Com.stComIn_DREAM_DP1_PTM_01/D[2] <-> COM TxPDO-Map Inputs/Data In 2
//     Serial_COM Inputs/GVL_Serial_Com.stComIn_DREAM_DP1_PTM_01/D[3] <-> COM TxPDO-Map Inputs/Data In 3
//     Serial_COM Inputs/GVL_Serial_Com.stComIn_DREAM_DP1_PTM_01/D[4] <-> COM TxPDO-Map Inputs/Data In 4
//     Serial_COM Inputs/GVL_Serial_Com.stComIn_DREAM_DP1_PTM_01/D[5] <-> COM TxPDO-Map Inputs/Data In 5
//     Serial_COM Inputs/GVL_Serial_Com.stComIn_DREAM_DP1_PTM_01/D[6] <-> COM TxPDO-Map Inputs/Data In 6
//     Serial_COM Inputs/GVL_Serial_Com.stComIn_DREAM_DP1_PTM_01/D[7] <-> COM TxPDO-Map Inputs/Data In 7
//     Serial_COM Inputs/GVL_Serial_Com.stComIn_DREAM_DP1_PTM_01/D[8] <-> COM TxPDO-Map Inputs/Data In 8
//     Serial_COM Inputs/GVL_Serial_Com.stComIn_DREAM_DP1_PTM_01/D[9] <-> COM TxPDO-Map Inputs/Data In 9
//     Serial_COM Inputs/GVL_Serial_Com.stComIn_DREAM_DP1_PTM_01/Status <-> COM TxPDO-Map Inputs/Status
//     Serial_COM Outputs/GVL_Serial_Com.stComOut_DREAM_DP1_PTM_01/Ctrl <-> COM RxPDO-Map Outputs/Ctrl
//     Serial_COM Outputs/GVL_Serial_Com.stComOut_DREAM_DP1_PTM_01/D[0] <-> COM RxPDO-Map Outputs/Data Out 0
//     Serial_COM Outputs/GVL_Serial_Com.stComOut_DREAM_DP1_PTM_01/D[10] <-> COM RxPDO-Map Outputs/Data Out 10
//     Serial_COM Outputs/GVL_Serial_Com.stComOut_DREAM_DP1_PTM_01/D[11] <-> COM RxPDO-Map Outputs/Data Out 11
//     Serial_COM Outputs/GVL_Serial_Com.stComOut_DREAM_DP1_PTM_01/D[12] <-> COM RxPDO-Map Outputs/Data Out 12
//     Serial_COM Outputs/GVL_Serial_Com.stComOut_DREAM_DP1_PTM_01/D[13] <-> COM RxPDO-Map Outputs/Data Out 13
//     Serial_COM Outputs/GVL_Serial_Com.stComOut_DREAM_DP1_PTM_01/D[14] <-> COM RxPDO-Map Outputs/Data Out 14
//     Serial_COM Outputs/GVL_Serial_Com.stComOut_DREAM_DP1_PTM_01/D[15] <-> COM RxPDO-Map Outputs/Data Out 15
//     Serial_COM Outputs/GVL_Serial_Com.stComOut_DREAM_DP1_PTM_01/D[16] <-> COM RxPDO-Map Outputs/Data Out 16
//     Serial_COM Outputs/GVL_Serial_Com.stComOut_DREAM_DP1_PTM_01/D[17] <-> COM RxPDO-Map Outputs/Data Out 17
//     Serial_COM Outputs/GVL_Serial_Com.stComOut_DREAM_DP1_PTM_01/D[18] <-> COM RxPDO-Map Outputs/Data Out 18
//     Serial_COM Outputs/GVL_Serial_Com.stComOut_DREAM_DP1_PTM_01/D[19] <-> COM RxPDO-Map Outputs/Data Out 19
//     Serial_COM Outputs/GVL_Serial_Com.stComOut_DREAM_DP1_PTM_01/D[1] <-> COM RxPDO-Map Outputs/Data Out 1
//     Serial_COM Outputs/GVL_Serial_Com.stComOut_DREAM_DP1_PTM_01/D[20] <-> COM RxPDO-Map Outputs/Data Out 20
//     Serial_COM Outputs/GVL_Serial_Com.stComOut_DREAM_DP1_PTM_01/D[21] <-> COM RxPDO-Map Outputs/Data Out 21
//     Serial_COM Outputs/GVL_Serial_Com.stComOut_DREAM_DP1_PTM_01/D[2] <-> COM RxPDO-Map Outputs/Data Out 2
//     Serial_COM Outputs/GVL_Serial_Com.stComOut_DREAM_DP1_PTM_01/D[3] <-> COM RxPDO-Map Outputs/Data Out 3
//     Serial_COM Outputs/GVL_Serial_Com.stComOut_DREAM_DP1_PTM_01/D[4] <-> COM RxPDO-Map Outputs/Data Out 4
//     Serial_COM Outputs/GVL_Serial_Com.stComOut_DREAM_DP1_PTM_01/D[5] <-> COM RxPDO-Map Outputs/Data Out 5
//     Serial_COM Outputs/GVL_Serial_Com.stComOut_DREAM_DP1_PTM_01/D[6] <-> COM RxPDO-Map Outputs/Data Out 6
//     Serial_COM Outputs/GVL_Serial_Com.stComOut_DREAM_DP1_PTM_01/D[7] <-> COM RxPDO-Map Outputs/Data Out 7
//     Serial_COM Outputs/GVL_Serial_Com.stComOut_DREAM_DP1_PTM_01/D[8] <-> COM RxPDO-Map Outputs/Data Out 8
//     Serial_COM Outputs/GVL_Serial_Com.stComOut_DREAM_DP1_PTM_01/D[9] <-> COM RxPDO-Map Outputs/Data Out 9
//   lcls_plc_dream_vac Instance <-> Device 1 (EtherCAT)/R20_DRL_03_CX0_EK1200/R20_DRL_03_E15_EL1122/K4S8_DRL_03_EK0_EK1100/K4S8_DRL_03_E19_EL1004
//     PlcTask Inputs/GVL_VAC_PUMPS.DREAM_DP1_PTM_01.i_xAtSpd <-> Channel 1/Input
//     PlcTask Inputs/GVL_VAC_PUMPS.DREAM_DP1_PTM_01.i_xFaultNC <-> Channel 3/Input
//     PlcTask Inputs/GVL_VAC_PUMPS.DREAM_DP1_PTM_01.i_xRemote <-> Channel 2/Input
//   lcls_plc_dream_vac Instance <-> Device 1 (EtherCAT)/R20_DRL_03_CX0_EK1200/R20_DRL_03_E15_EL1122/K4S8_DRL_03_EK0_EK1100/K4S8_DRL_03_E1_EL2624
//     PlcTask Outputs/GVL_VAC_GAUGES.DREAM_DP1_GHC_01.q_xHV_DIS <-> Channel 2/Output
//     PlcTask Outputs/GVL_VAC_GAUGES.DREAM_DP2_GHC_01.q_xHV_DIS <-> Channel 3/Output
//     PlcTask Outputs/GVL_VAC_GAUGES.DREAM_DP3_GHC_01.q_xHV_DIS <-> Channel 4/Output
//     PlcTask Outputs/GVL_VAC_GAUGES.DREAM_NC_GCC_01.q_xHV_DIS <-> Channel 1/Output
//   lcls_plc_dream_vac Instance <-> Device 1 (EtherCAT)/R20_DRL_03_CX0_EK1200/R20_DRL_03_E15_EL1122/K4S8_DRL_03_EK0_EK1100/K4S8_DRL_03_E20_EL2004
//     PlcTask Outputs/GVL_VAC_PUMPS.DREAM_DP1_PTM_01.q_PumpingStation <-> Channel 3/Output
//     PlcTask Outputs/GVL_VAC_PUMPS.DREAM_DP1_PTM_01.q_RunDO <-> Channel 1/Output
//     PlcTask Outputs/GVL_VAC_PUMPS.DREAM_DP1_PTM_01.q_xRemote <-> Channel 2/Output
//   lcls_plc_dream_vac Instance <-> Device 1 (EtherCAT)/R20_DRL_03_CX0_EK1200/R20_DRL_03_E15_EL1122/K4S8_DRL_03_EK0_EK1100/K4S8_DRL_03_E21_EL3052
//     PlcTask Inputs/GVL_FWM.fbCoilFlowMeter.iRaw <-> AI Standard Channel 1/Value
//   lcls_plc_dream_vac Instance <-> Device 1 (EtherCAT)/R20_DRL_03_CX0_EK1200/R20_DRL_03_E15_EL1122/K4S8_DRL_03_EK0_EK1100/K4S8_DRL_03_E4_EL1084
//     PlcTask Inputs/GVL_VAC_GAUGES.DREAM_DP1_GHC_01.i_xHV_ON <-> Channel 4/Input
//     PlcTask Inputs/GVL_VAC_GAUGES.DREAM_DP2_GHC_01.i_xHV_ON <-> Channel 1/Input
//     PlcTask Inputs/GVL_VAC_GAUGES.DREAM_DP3_GHC_01.i_xHV_ON <-> Channel 2/Input
//     PlcTask Inputs/GVL_VAC_GAUGES.DREAM_NC_GCC_01.i_xHV_ON <-> Channel 3/Input
//   lcls_plc_dream_vac Instance <-> Device 1 (EtherCAT)/R20_DRL_03_CX0_EK1200/R20_DRL_03_E15_EL1122/K4S8_DRL_03_EK0_EK1100/K4S8_DRL_03_E5_EL3174-0002
//     PlcTask Inputs/GVL_VAC_GAUGES.DREAM_DP1_GHC_01.i_iPRESS_R <-> AI Standard Channel 2/Value
//     PlcTask Inputs/GVL_VAC_GAUGES.DREAM_DP2_GHC_01.i_iPRESS_R <-> AI Standard Channel 3/Value
//     PlcTask Inputs/GVL_VAC_GAUGES.DREAM_DP3_GHC_01.i_iPRESS_R <-> AI Standard Channel 4/Value
//     PlcTask Inputs/GVL_VAC_GAUGES.DREAM_NC_GCC_01.i_iPRESS_R <-> AI Standard Channel 1/Value
//   lcls_plc_dream_vac Instance <-> Device 1 (EtherCAT)/R20_DRL_03_CX0_EK1200/R20_DRL_03_E15_EL1122/K4S8_DRL_03_EK0_EK1100/K4S8_DRL_03_E6_EL3174-0002
//     PlcTask Inputs/GVL_VAC_GAUGES.DREAM_DP1_GPI_01.i_iPRESS_R <-> AI Standard Channel 2/Value
//     PlcTask Inputs/GVL_VAC_GAUGES.DREAM_NC_GPI_01.i_iPRESS_R <-> AI Standard Channel 1/Value
//   lcls_plc_dream_vac Instance <-> Device 1 (EtherCAT)/R20_DRL_03_CX0_EK1200/R20_DRL_03_E15_EL1122/K4S8_DRL_04_EK0_EK1100/K4S8_DRL_04_E10_EL1004
//     PlcTask Inputs/GVL_VAC_VALVES.DREAM_ROUGH2_VRC_02.i_xClsLS <-> Channel 2/Input
//     PlcTask Inputs/GVL_VAC_VALVES.DREAM_ROUGH2_VRC_02.i_xOpnLS <-> Channel 1/Input
//   lcls_plc_dream_vac Instance <-> Device 1 (EtherCAT)/R20_DRL_03_CX0_EK1200/R20_DRL_03_E15_EL1122/K4S8_DRL_04_EK0_EK1100/K4S8_DRL_04_E11_EL2004
//     PlcTask Outputs/GVL_VAC_VALVES.DREAM_ROUGH1_VRC_01.q_xOPN_DO <-> Channel 1/Output
//     PlcTask Outputs/GVL_VAC_VALVES.DREAM_ROUGH2_VRC_01.q_xOPN_DO <-> Channel 2/Output
//     PlcTask Outputs/GVL_VAC_VALVES.DREAM_ROUGH2_VRC_02.q_xOPN_DO <-> Channel 3/Output
//   lcls_plc_dream_vac Instance <-> Device 1 (EtherCAT)/R20_DRL_03_CX0_EK1200/R20_DRL_03_E15_EL1122/K4S8_DRL_04_EK0_EK1100/K4S8_DRL_04_E14_EL2624
//     PlcTask Outputs/GVL_PLC_Interface.bCoilPS_ILK <-> Channel 3/Output
//     PlcTask Outputs/GVL_PLC_Interface.bHighVoltageSafteyLoopEnable <-> Channel 4/Output
//     PlcTask Outputs/GVL_VAC_GAUGES.DREAM_CAT1_GHC_01.q_xHV_DIS <-> Channel 1/Output
//     PlcTask Outputs/GVL_VAC_GAUGES.DREAM_CAT2_GHC_01.q_xHV_DIS <-> Channel 2/Output
//   lcls_plc_dream_vac Instance <-> Device 1 (EtherCAT)/R20_DRL_03_CX0_EK1200/R20_DRL_03_E15_EL1122/K4S8_DRL_04_EK0_EK1100/K4S8_DRL_04_E15_EL1084
//     PlcTask Inputs/GVL_VAC_GAUGES.DREAM_CAT1_GHC_01.i_xHV_ON <-> Channel 1/Input
//     PlcTask Inputs/GVL_VAC_GAUGES.DREAM_CAT2_GHC_01.i_xHV_ON <-> Channel 2/Input
//   lcls_plc_dream_vac Instance <-> Device 1 (EtherCAT)/R20_DRL_03_CX0_EK1200/R20_DRL_03_E15_EL1122/K4S8_DRL_04_EK0_EK1100/K4S8_DRL_04_E16_EL3174-0002
//     PlcTask Inputs/GVL_VAC_GAUGES.DREAM_CAT1_GHC_01.i_iPRESS_R <-> AI Standard Channel 2/Value
//     PlcTask Inputs/GVL_VAC_GAUGES.DREAM_CAT2_GHC_01.i_iPRESS_R <-> AI Standard Channel 3/Value
//     PlcTask Inputs/GVL_VAC_GAUGES.DREAM_MC_GPI_01.i_iPRESS_R <-> AI Standard Channel 1/Value
//   lcls_plc_dream_vac Instance <-> Device 1 (EtherCAT)/R20_DRL_03_CX0_EK1200/R20_DRL_03_E15_EL1122/K4S8_DRL_04_EK0_EK1100/K4S8_DRL_04_E17_EL6001
//     Serial_COM Inputs/GVL_Serial_Com.stComIn_DREAM_ROUGH2_PTM_02/D[0] <-> COM Inputs/Data In 0
//     Serial_COM Inputs/GVL_Serial_Com.stComIn_DREAM_ROUGH2_PTM_02/D[10] <-> COM Inputs/Data In 10
//     Serial_COM Inputs/GVL_Serial_Com.stComIn_DREAM_ROUGH2_PTM_02/D[11] <-> COM Inputs/Data In 11
//     Serial_COM Inputs/GVL_Serial_Com.stComIn_DREAM_ROUGH2_PTM_02/D[12] <-> COM Inputs/Data In 12
//     Serial_COM Inputs/GVL_Serial_Com.stComIn_DREAM_ROUGH2_PTM_02/D[13] <-> COM Inputs/Data In 13
//     Serial_COM Inputs/GVL_Serial_Com.stComIn_DREAM_ROUGH2_PTM_02/D[14] <-> COM Inputs/Data In 14
//     Serial_COM Inputs/GVL_Serial_Com.stComIn_DREAM_ROUGH2_PTM_02/D[15] <-> COM Inputs/Data In 15
//     Serial_COM Inputs/GVL_Serial_Com.stComIn_DREAM_ROUGH2_PTM_02/D[16] <-> COM Inputs/Data In 16
//     Serial_COM Inputs/GVL_Serial_Com.stComIn_DREAM_ROUGH2_PTM_02/D[17] <-> COM Inputs/Data In 17
//     Serial_COM Inputs/GVL_Serial_Com.stComIn_DREAM_ROUGH2_PTM_02/D[18] <-> COM Inputs/Data In 18
//     Serial_COM Inputs/GVL_Serial_Com.stComIn_DREAM_ROUGH2_PTM_02/D[19] <-> COM Inputs/Data In 19
//     Serial_COM Inputs/GVL_Serial_Com.stComIn_DREAM_ROUGH2_PTM_02/D[1] <-> COM Inputs/Data In 1
//     Serial_COM Inputs/GVL_Serial_Com.stComIn_DREAM_ROUGH2_PTM_02/D[20] <-> COM Inputs/Data In 20
//     Serial_COM Inputs/GVL_Serial_Com.stComIn_DREAM_ROUGH2_PTM_02/D[21] <-> COM Inputs/Data In 21
//     Serial_COM Inputs/GVL_Serial_Com.stComIn_DREAM_ROUGH2_PTM_02/D[2] <-> COM Inputs/Data In 2
//     Serial_COM Inputs/GVL_Serial_Com.stComIn_DREAM_ROUGH2_PTM_02/D[3] <-> COM Inputs/Data In 3
//     Serial_COM Inputs/GVL_Serial_Com.stComIn_DREAM_ROUGH2_PTM_02/D[4] <-> COM Inputs/Data In 4
//     Serial_COM Inputs/GVL_Serial_Com.stComIn_DREAM_ROUGH2_PTM_02/D[5] <-> COM Inputs/Data In 5
//     Serial_COM Inputs/GVL_Serial_Com.stComIn_DREAM_ROUGH2_PTM_02/D[6] <-> COM Inputs/Data In 6
//     Serial_COM Inputs/GVL_Serial_Com.stComIn_DREAM_ROUGH2_PTM_02/D[7] <-> COM Inputs/Data In 7
//     Serial_COM Inputs/GVL_Serial_Com.stComIn_DREAM_ROUGH2_PTM_02/D[8] <-> COM Inputs/Data In 8
//     Serial_COM Inputs/GVL_Serial_Com.stComIn_DREAM_ROUGH2_PTM_02/D[9] <-> COM Inputs/Data In 9
//     Serial_COM Inputs/GVL_Serial_Com.stComIn_DREAM_ROUGH2_PTM_02/Status <-> COM Inputs/Status
//     Serial_COM Outputs/GVL_Serial_Com.stComOut_DREAM_ROUGH2_PTM_02/Ctrl <-> COM Outputs/Ctrl
//     Serial_COM Outputs/GVL_Serial_Com.stComOut_DREAM_ROUGH2_PTM_02/D[0] <-> COM Outputs/Data Out 0
//     Serial_COM Outputs/GVL_Serial_Com.stComOut_DREAM_ROUGH2_PTM_02/D[10] <-> COM Outputs/Data Out 10
//     Serial_COM Outputs/GVL_Serial_Com.stComOut_DREAM_ROUGH2_PTM_02/D[11] <-> COM Outputs/Data Out 11
//     Serial_COM Outputs/GVL_Serial_Com.stComOut_DREAM_ROUGH2_PTM_02/D[12] <-> COM Outputs/Data Out 12
//     Serial_COM Outputs/GVL_Serial_Com.stComOut_DREAM_ROUGH2_PTM_02/D[13] <-> COM Outputs/Data Out 13
//     Serial_COM Outputs/GVL_Serial_Com.stComOut_DREAM_ROUGH2_PTM_02/D[14] <-> COM Outputs/Data Out 14
//     Serial_COM Outputs/GVL_Serial_Com.stComOut_DREAM_ROUGH2_PTM_02/D[15] <-> COM Outputs/Data Out 15
//     Serial_COM Outputs/GVL_Serial_Com.stComOut_DREAM_ROUGH2_PTM_02/D[16] <-> COM Outputs/Data Out 16
//     Serial_COM Outputs/GVL_Serial_Com.stComOut_DREAM_ROUGH2_PTM_02/D[17] <-> COM Outputs/Data Out 17
//     Serial_COM Outputs/GVL_Serial_Com.stComOut_DREAM_ROUGH2_PTM_02/D[18] <-> COM Outputs/Data Out 18
//     Serial_COM Outputs/GVL_Serial_Com.stComOut_DREAM_ROUGH2_PTM_02/D[19] <-> COM Outputs/Data Out 19
//     Serial_COM Outputs/GVL_Serial_Com.stComOut_DREAM_ROUGH2_PTM_02/D[1] <-> COM Outputs/Data Out 1
//     Serial_COM Outputs/GVL_Serial_Com.stComOut_DREAM_ROUGH2_PTM_02/D[20] <-> COM Outputs/Data Out 20
//     Serial_COM Outputs/GVL_Serial_Com.stComOut_DREAM_ROUGH2_PTM_02/D[21] <-> COM Outputs/Data Out 21
//     Serial_COM Outputs/GVL_Serial_Com.stComOut_DREAM_ROUGH2_PTM_02/D[2] <-> COM Outputs/Data Out 2
//     Serial_COM Outputs/GVL_Serial_Com.stComOut_DREAM_ROUGH2_PTM_02/D[3] <-> COM Outputs/Data Out 3
//     Serial_COM Outputs/GVL_Serial_Com.stComOut_DREAM_ROUGH2_PTM_02/D[4] <-> COM Outputs/Data Out 4
//     Serial_COM Outputs/GVL_Serial_Com.stComOut_DREAM_ROUGH2_PTM_02/D[5] <-> COM Outputs/Data Out 5
//     Serial_COM Outputs/GVL_Serial_Com.stComOut_DREAM_ROUGH2_PTM_02/D[6] <-> COM Outputs/Data Out 6
//     Serial_COM Outputs/GVL_Serial_Com.stComOut_DREAM_ROUGH2_PTM_02/D[7] <-> COM Outputs/Data Out 7
//     Serial_COM Outputs/GVL_Serial_Com.stComOut_DREAM_ROUGH2_PTM_02/D[8] <-> COM Outputs/Data Out 8
//     Serial_COM Outputs/GVL_Serial_Com.stComOut_DREAM_ROUGH2_PTM_02/D[9] <-> COM Outputs/Data Out 9
//   lcls_plc_dream_vac Instance <-> Device 1 (EtherCAT)/R20_DRL_03_CX0_EK1200/R20_DRL_03_E15_EL1122/K4S8_DRL_04_EK0_EK1100/K4S8_DRL_04_E1_EL1004
//     PlcTask Inputs/GVL_VAC_VALVES.DREAM_CAT1_VRC_01.i_xClsLS <-> Channel 2/Input
//     PlcTask Inputs/GVL_VAC_VALVES.DREAM_CAT1_VRC_01.i_xOpnLS <-> Channel 1/Input
//   lcls_plc_dream_vac Instance <-> Device 1 (EtherCAT)/R20_DRL_03_CX0_EK1200/R20_DRL_03_E15_EL1122/K4S8_DRL_04_EK0_EK1100/K4S8_DRL_04_E2_EL2004
//     PlcTask Outputs/GVL_VAC_VALVES.DREAM_CAT1_VRC_01.q_xOPN_DO <-> Channel 1/Output
//   lcls_plc_dream_vac Instance <-> Device 1 (EtherCAT)/R20_DRL_03_CX0_EK1200/R20_DRL_03_E15_EL1122/K4S8_DRL_04_EK0_EK1100/K4S8_DRL_04_E3_EL1004
//     PlcTask Inputs/GVL_VAC_PUMPS.DREAM_CAT1_PTM_01.i_xAtSpd <-> Channel 4/Input
//     PlcTask Inputs/GVL_VAC_PUMPS.DREAM_CAT1_PTM_01.i_xFaultNC <-> Channel 3/Input
//     PlcTask Inputs/GVL_VAC_PUMPS.DREAM_ROUGH2_PTM_01.i_xAtSpd <-> Channel 2/Input
//     PlcTask Inputs/GVL_VAC_PUMPS.DREAM_ROUGH2_PTM_01.i_xFaultNC <-> Channel 1/Input
//   lcls_plc_dream_vac Instance <-> Device 1 (EtherCAT)/R20_DRL_03_CX0_EK1200/R20_DRL_03_E15_EL1122/K4S8_DRL_04_EK0_EK1100/K4S8_DRL_04_E4_EL1004
//     PlcTask Inputs/GVL_VAC_PUMPS.DREAM_CAT2_PTM_01.i_xAtSpd <-> Channel 2/Input
//     PlcTask Inputs/GVL_VAC_PUMPS.DREAM_CAT2_PTM_01.i_xFaultNC <-> Channel 1/Input
//     PlcTask Inputs/GVL_VAC_PUMPS.DREAM_ROUGH2_PTM_02.i_xAtSpd <-> Channel 4/Input
//     PlcTask Inputs/GVL_VAC_PUMPS.DREAM_ROUGH2_PTM_02.i_xFaultNC <-> Channel 3/Input
//   lcls_plc_dream_vac Instance <-> Device 1 (EtherCAT)/R20_DRL_03_CX0_EK1200/R20_DRL_03_E15_EL1122/K4S8_DRL_04_EK0_EK1100/K4S8_DRL_04_E5_EL2794
//     PlcTask Outputs/GVL_VAC_PUMPS.DREAM_CAT1_PTM_01.q_RunDO <-> Channel 2/Output
//     PlcTask Outputs/GVL_VAC_PUMPS.DREAM_CAT2_PTM_01.q_RunDO <-> Channel 3/Output
//     PlcTask Outputs/GVL_VAC_PUMPS.DREAM_ROUGH2_PTM_01.q_RunDO <-> Channel 1/Output
//     PlcTask Outputs/GVL_VAC_PUMPS.DREAM_ROUGH2_PTM_02.q_RunDO <-> Channel 4/Output
//   lcls_plc_dream_vac Instance <-> Device 1 (EtherCAT)/R20_DRL_03_CX0_EK1200/R20_DRL_03_E15_EL1122/K4S8_DRL_04_EK0_EK1100/K4S8_DRL_04_E6_EL6001
//     Serial_COM Inputs/GVL_Serial_Com.stComIn_DREAM_ROUGH2_PTM_01/D[0] <-> COM Inputs/Data In 0
//     Serial_COM Inputs/GVL_Serial_Com.stComIn_DREAM_ROUGH2_PTM_01/D[10] <-> COM Inputs/Data In 10
//     Serial_COM Inputs/GVL_Serial_Com.stComIn_DREAM_ROUGH2_PTM_01/D[11] <-> COM Inputs/Data In 11
//     Serial_COM Inputs/GVL_Serial_Com.stComIn_DREAM_ROUGH2_PTM_01/D[12] <-> COM Inputs/Data In 12
//     Serial_COM Inputs/GVL_Serial_Com.stComIn_DREAM_ROUGH2_PTM_01/D[13] <-> COM Inputs/Data In 13
//     Serial_COM Inputs/GVL_Serial_Com.stComIn_DREAM_ROUGH2_PTM_01/D[14] <-> COM Inputs/Data In 14
//     Serial_COM Inputs/GVL_Serial_Com.stComIn_DREAM_ROUGH2_PTM_01/D[15] <-> COM Inputs/Data In 15
//     Serial_COM Inputs/GVL_Serial_Com.stComIn_DREAM_ROUGH2_PTM_01/D[16] <-> COM Inputs/Data In 16
//     Serial_COM Inputs/GVL_Serial_Com.stComIn_DREAM_ROUGH2_PTM_01/D[17] <-> COM Inputs/Data In 17
//     Serial_COM Inputs/GVL_Serial_Com.stComIn_DREAM_ROUGH2_PTM_01/D[18] <-> COM Inputs/Data In 18
//     Serial_COM Inputs/GVL_Serial_Com.stComIn_DREAM_ROUGH2_PTM_01/D[19] <-> COM Inputs/Data In 19
//     Serial_COM Inputs/GVL_Serial_Com.stComIn_DREAM_ROUGH2_PTM_01/D[1] <-> COM Inputs/Data In 1
//     Serial_COM Inputs/GVL_Serial_Com.stComIn_DREAM_ROUGH2_PTM_01/D[20] <-> COM Inputs/Data In 20
//     Serial_COM Inputs/GVL_Serial_Com.stComIn_DREAM_ROUGH2_PTM_01/D[21] <-> COM Inputs/Data In 21
//     Serial_COM Inputs/GVL_Serial_Com.stComIn_DREAM_ROUGH2_PTM_01/D[2] <-> COM Inputs/Data In 2
//     Serial_COM Inputs/GVL_Serial_Com.stComIn_DREAM_ROUGH2_PTM_01/D[3] <-> COM Inputs/Data In 3
//     Serial_COM Inputs/GVL_Serial_Com.stComIn_DREAM_ROUGH2_PTM_01/D[4] <-> COM Inputs/Data In 4
//     Serial_COM Inputs/GVL_Serial_Com.stComIn_DREAM_ROUGH2_PTM_01/D[5] <-> COM Inputs/Data In 5
//     Serial_COM Inputs/GVL_Serial_Com.stComIn_DREAM_ROUGH2_PTM_01/D[6] <-> COM Inputs/Data In 6
//     Serial_COM Inputs/GVL_Serial_Com.stComIn_DREAM_ROUGH2_PTM_01/D[7] <-> COM Inputs/Data In 7
//     Serial_COM Inputs/GVL_Serial_Com.stComIn_DREAM_ROUGH2_PTM_01/D[8] <-> COM Inputs/Data In 8
//     Serial_COM Inputs/GVL_Serial_Com.stComIn_DREAM_ROUGH2_PTM_01/D[9] <-> COM Inputs/Data In 9
//     Serial_COM Inputs/GVL_Serial_Com.stComIn_DREAM_ROUGH2_PTM_01/Status <-> COM Inputs/Status
//     Serial_COM Outputs/GVL_Serial_Com.stComOut_DREAM_ROUGH2_PTM_01/Ctrl <-> COM Outputs/Ctrl
//     Serial_COM Outputs/GVL_Serial_Com.stComOut_DREAM_ROUGH2_PTM_01/D[0] <-> COM Outputs/Data Out 0
//     Serial_COM Outputs/GVL_Serial_Com.stComOut_DREAM_ROUGH2_PTM_01/D[10] <-> COM Outputs/Data Out 10
//     Serial_COM Outputs/GVL_Serial_Com.stComOut_DREAM_ROUGH2_PTM_01/D[11] <-> COM Outputs/Data Out 11
//     Serial_COM Outputs/GVL_Serial_Com.stComOut_DREAM_ROUGH2_PTM_01/D[12] <-> COM Outputs/Data Out 12
//     Serial_COM Outputs/GVL_Serial_Com.stComOut_DREAM_ROUGH2_PTM_01/D[13] <-> COM Outputs/Data Out 13
//     Serial_COM Outputs/GVL_Serial_Com.stComOut_DREAM_ROUGH2_PTM_01/D[14] <-> COM Outputs/Data Out 14
//     Serial_COM Outputs/GVL_Serial_Com.stComOut_DREAM_ROUGH2_PTM_01/D[15] <-> COM Outputs/Data Out 15
//     Serial_COM Outputs/GVL_Serial_Com.stComOut_DREAM_ROUGH2_PTM_01/D[16] <-> COM Outputs/Data Out 16
//     Serial_COM Outputs/GVL_Serial_Com.stComOut_DREAM_ROUGH2_PTM_01/D[17] <-> COM Outputs/Data Out 17
//     Serial_COM Outputs/GVL_Serial_Com.stComOut_DREAM_ROUGH2_PTM_01/D[18] <-> COM Outputs/Data Out 18
//     Serial_COM Outputs/GVL_Serial_Com.stComOut_DREAM_ROUGH2_PTM_01/D[19] <-> COM Outputs/Data Out 19
//     Serial_COM Outputs/GVL_Serial_Com.stComOut_DREAM_ROUGH2_PTM_01/D[1] <-> COM Outputs/Data Out 1
//     Serial_COM Outputs/GVL_Serial_Com.stComOut_DREAM_ROUGH2_PTM_01/D[20] <-> COM Outputs/Data Out 20
//     Serial_COM Outputs/GVL_Serial_Com.stComOut_DREAM_ROUGH2_PTM_01/D[21] <-> COM Outputs/Data Out 21
//     Serial_COM Outputs/GVL_Serial_Com.stComOut_DREAM_ROUGH2_PTM_01/D[2] <-> COM Outputs/Data Out 2
//     Serial_COM Outputs/GVL_Serial_Com.stComOut_DREAM_ROUGH2_PTM_01/D[3] <-> COM Outputs/Data Out 3
//     Serial_COM Outputs/GVL_Serial_Com.stComOut_DREAM_ROUGH2_PTM_01/D[4] <-> COM Outputs/Data Out 4
//     Serial_COM Outputs/GVL_Serial_Com.stComOut_DREAM_ROUGH2_PTM_01/D[5] <-> COM Outputs/Data Out 5
//     Serial_COM Outputs/GVL_Serial_Com.stComOut_DREAM_ROUGH2_PTM_01/D[6] <-> COM Outputs/Data Out 6
//     Serial_COM Outputs/GVL_Serial_Com.stComOut_DREAM_ROUGH2_PTM_01/D[7] <-> COM Outputs/Data Out 7
//     Serial_COM Outputs/GVL_Serial_Com.stComOut_DREAM_ROUGH2_PTM_01/D[8] <-> COM Outputs/Data Out 8
//     Serial_COM Outputs/GVL_Serial_Com.stComOut_DREAM_ROUGH2_PTM_01/D[9] <-> COM Outputs/Data Out 9
//   lcls_plc_dream_vac Instance <-> Device 1 (EtherCAT)/R20_DRL_03_CX0_EK1200/R20_DRL_03_E15_EL1122/K4S8_DRL_04_EK0_EK1100/K4S8_DRL_04_E7_EL6001
//     Serial_COM Inputs/GVL_Serial_Com.stComIn_DREAM_CAT1_PTM_01/D[0] <-> COM Inputs/Data In 0
//     Serial_COM Inputs/GVL_Serial_Com.stComIn_DREAM_CAT1_PTM_01/D[10] <-> COM Inputs/Data In 10
//     Serial_COM Inputs/GVL_Serial_Com.stComIn_DREAM_CAT1_PTM_01/D[11] <-> COM Inputs/Data In 11
//     Serial_COM Inputs/GVL_Serial_Com.stComIn_DREAM_CAT1_PTM_01/D[12] <-> COM Inputs/Data In 12
//     Serial_COM Inputs/GVL_Serial_Com.stComIn_DREAM_CAT1_PTM_01/D[13] <-> COM Inputs/Data In 13
//     Serial_COM Inputs/GVL_Serial_Com.stComIn_DREAM_CAT1_PTM_01/D[14] <-> COM Inputs/Data In 14
//     Serial_COM Inputs/GVL_Serial_Com.stComIn_DREAM_CAT1_PTM_01/D[15] <-> COM Inputs/Data In 15
//     Serial_COM Inputs/GVL_Serial_Com.stComIn_DREAM_CAT1_PTM_01/D[16] <-> COM Inputs/Data In 16
//     Serial_COM Inputs/GVL_Serial_Com.stComIn_DREAM_CAT1_PTM_01/D[17] <-> COM Inputs/Data In 17
//     Serial_COM Inputs/GVL_Serial_Com.stComIn_DREAM_CAT1_PTM_01/D[18] <-> COM Inputs/Data In 18
//     Serial_COM Inputs/GVL_Serial_Com.stComIn_DREAM_CAT1_PTM_01/D[19] <-> COM Inputs/Data In 19
//     Serial_COM Inputs/GVL_Serial_Com.stComIn_DREAM_CAT1_PTM_01/D[1] <-> COM Inputs/Data In 1
//     Serial_COM Inputs/GVL_Serial_Com.stComIn_DREAM_CAT1_PTM_01/D[20] <-> COM Inputs/Data In 20
//     Serial_COM Inputs/GVL_Serial_Com.stComIn_DREAM_CAT1_PTM_01/D[21] <-> COM Inputs/Data In 21
//     Serial_COM Inputs/GVL_Serial_Com.stComIn_DREAM_CAT1_PTM_01/D[2] <-> COM Inputs/Data In 2
//     Serial_COM Inputs/GVL_Serial_Com.stComIn_DREAM_CAT1_PTM_01/D[3] <-> COM Inputs/Data In 3
//     Serial_COM Inputs/GVL_Serial_Com.stComIn_DREAM_CAT1_PTM_01/D[4] <-> COM Inputs/Data In 4
//     Serial_COM Inputs/GVL_Serial_Com.stComIn_DREAM_CAT1_PTM_01/D[5] <-> COM Inputs/Data In 5
//     Serial_COM Inputs/GVL_Serial_Com.stComIn_DREAM_CAT1_PTM_01/D[6] <-> COM Inputs/Data In 6
//     Serial_COM Inputs/GVL_Serial_Com.stComIn_DREAM_CAT1_PTM_01/D[7] <-> COM Inputs/Data In 7
//     Serial_COM Inputs/GVL_Serial_Com.stComIn_DREAM_CAT1_PTM_01/D[8] <-> COM Inputs/Data In 8
//     Serial_COM Inputs/GVL_Serial_Com.stComIn_DREAM_CAT1_PTM_01/D[9] <-> COM Inputs/Data In 9
//     Serial_COM Inputs/GVL_Serial_Com.stComIn_DREAM_CAT1_PTM_01/Status <-> COM Inputs/Status
//     Serial_COM Outputs/GVL_Serial_Com.stComOut_DREAM_CAT1_PTM_01/Ctrl <-> COM Outputs/Ctrl
//     Serial_COM Outputs/GVL_Serial_Com.stComOut_DREAM_CAT1_PTM_01/D[0] <-> COM Outputs/Data Out 0
//     Serial_COM Outputs/GVL_Serial_Com.stComOut_DREAM_CAT1_PTM_01/D[10] <-> COM Outputs/Data Out 10
//     Serial_COM Outputs/GVL_Serial_Com.stComOut_DREAM_CAT1_PTM_01/D[11] <-> COM Outputs/Data Out 11
//     Serial_COM Outputs/GVL_Serial_Com.stComOut_DREAM_CAT1_PTM_01/D[12] <-> COM Outputs/Data Out 12
//     Serial_COM Outputs/GVL_Serial_Com.stComOut_DREAM_CAT1_PTM_01/D[13] <-> COM Outputs/Data Out 13
//     Serial_COM Outputs/GVL_Serial_Com.stComOut_DREAM_CAT1_PTM_01/D[14] <-> COM Outputs/Data Out 14
//     Serial_COM Outputs/GVL_Serial_Com.stComOut_DREAM_CAT1_PTM_01/D[15] <-> COM Outputs/Data Out 15
//     Serial_COM Outputs/GVL_Serial_Com.stComOut_DREAM_CAT1_PTM_01/D[16] <-> COM Outputs/Data Out 16
//     Serial_COM Outputs/GVL_Serial_Com.stComOut_DREAM_CAT1_PTM_01/D[17] <-> COM Outputs/Data Out 17
//     Serial_COM Outputs/GVL_Serial_Com.stComOut_DREAM_CAT1_PTM_01/D[18] <-> COM Outputs/Data Out 18
//     Serial_COM Outputs/GVL_Serial_Com.stComOut_DREAM_CAT1_PTM_01/D[19] <-> COM Outputs/Data Out 19
//     Serial_COM Outputs/GVL_Serial_Com.stComOut_DREAM_CAT1_PTM_01/D[1] <-> COM Outputs/Data Out 1
//     Serial_COM Outputs/GVL_Serial_Com.stComOut_DREAM_CAT1_PTM_01/D[20] <-> COM Outputs/Data Out 20
//     Serial_COM Outputs/GVL_Serial_Com.stComOut_DREAM_CAT1_PTM_01/D[21] <-> COM Outputs/Data Out 21
//     Serial_COM Outputs/GVL_Serial_Com.stComOut_DREAM_CAT1_PTM_01/D[2] <-> COM Outputs/Data Out 2
//     Serial_COM Outputs/GVL_Serial_Com.stComOut_DREAM_CAT1_PTM_01/D[3] <-> COM Outputs/Data Out 3
//     Serial_COM Outputs/GVL_Serial_Com.stComOut_DREAM_CAT1_PTM_01/D[4] <-> COM Outputs/Data Out 4
//     Serial_COM Outputs/GVL_Serial_Com.stComOut_DREAM_CAT1_PTM_01/D[5] <-> COM Outputs/Data Out 5
//     Serial_COM Outputs/GVL_Serial_Com.stComOut_DREAM_CAT1_PTM_01/D[6] <-> COM Outputs/Data Out 6
//     Serial_COM Outputs/GVL_Serial_Com.stComOut_DREAM_CAT1_PTM_01/D[7] <-> COM Outputs/Data Out 7
//     Serial_COM Outputs/GVL_Serial_Com.stComOut_DREAM_CAT1_PTM_01/D[8] <-> COM Outputs/Data Out 8
//     Serial_COM Outputs/GVL_Serial_Com.stComOut_DREAM_CAT1_PTM_01/D[9] <-> COM Outputs/Data Out 9
//   lcls_plc_dream_vac Instance <-> Device 1 (EtherCAT)/R20_DRL_03_CX0_EK1200/R20_DRL_03_E15_EL1122/K4S8_DRL_04_EK0_EK1100/K4S8_DRL_04_E8_EL6001
//     Serial_COM Inputs/GVL_Serial_Com.stComIn_DREAM_CAT2_PTM_01/D[0] <-> COM Inputs/Data In 0
//     Serial_COM Inputs/GVL_Serial_Com.stComIn_DREAM_CAT2_PTM_01/D[10] <-> COM Inputs/Data In 10
//     Serial_COM Inputs/GVL_Serial_Com.stComIn_DREAM_CAT2_PTM_01/D[11] <-> COM Inputs/Data In 11
//     Serial_COM Inputs/GVL_Serial_Com.stComIn_DREAM_CAT2_PTM_01/D[12] <-> COM Inputs/Data In 12
//     Serial_COM Inputs/GVL_Serial_Com.stComIn_DREAM_CAT2_PTM_01/D[13] <-> COM Inputs/Data In 13
//     Serial_COM Inputs/GVL_Serial_Com.stComIn_DREAM_CAT2_PTM_01/D[14] <-> COM Inputs/Data In 14
//     Serial_COM Inputs/GVL_Serial_Com.stComIn_DREAM_CAT2_PTM_01/D[15] <-> COM Inputs/Data In 15
//     Serial_COM Inputs/GVL_Serial_Com.stComIn_DREAM_CAT2_PTM_01/D[16] <-> COM Inputs/Data In 16
//     Serial_COM Inputs/GVL_Serial_Com.stComIn_DREAM_CAT2_PTM_01/D[17] <-> COM Inputs/Data In 17
//     Serial_COM Inputs/GVL_Serial_Com.stComIn_DREAM_CAT2_PTM_01/D[18] <-> COM Inputs/Data In 18
//     Serial_COM Inputs/GVL_Serial_Com.stComIn_DREAM_CAT2_PTM_01/D[19] <-> COM Inputs/Data In 19
//     Serial_COM Inputs/GVL_Serial_Com.stComIn_DREAM_CAT2_PTM_01/D[1] <-> COM Inputs/Data In 1
//     Serial_COM Inputs/GVL_Serial_Com.stComIn_DREAM_CAT2_PTM_01/D[20] <-> COM Inputs/Data In 20
//     Serial_COM Inputs/GVL_Serial_Com.stComIn_DREAM_CAT2_PTM_01/D[21] <-> COM Inputs/Data In 21
//     Serial_COM Inputs/GVL_Serial_Com.stComIn_DREAM_CAT2_PTM_01/D[2] <-> COM Inputs/Data In 2
//     Serial_COM Inputs/GVL_Serial_Com.stComIn_DREAM_CAT2_PTM_01/D[3] <-> COM Inputs/Data In 3
//     Serial_COM Inputs/GVL_Serial_Com.stComIn_DREAM_CAT2_PTM_01/D[4] <-> COM Inputs/Data In 4
//     Serial_COM Inputs/GVL_Serial_Com.stComIn_DREAM_CAT2_PTM_01/D[5] <-> COM Inputs/Data In 5
//     Serial_COM Inputs/GVL_Serial_Com.stComIn_DREAM_CAT2_PTM_01/D[6] <-> COM Inputs/Data In 6
//     Serial_COM Inputs/GVL_Serial_Com.stComIn_DREAM_CAT2_PTM_01/D[7] <-> COM Inputs/Data In 7
//     Serial_COM Inputs/GVL_Serial_Com.stComIn_DREAM_CAT2_PTM_01/D[8] <-> COM Inputs/Data In 8
//     Serial_COM Inputs/GVL_Serial_Com.stComIn_DREAM_CAT2_PTM_01/D[9] <-> COM Inputs/Data In 9
//     Serial_COM Inputs/GVL_Serial_Com.stComIn_DREAM_CAT2_PTM_01/Status <-> COM Inputs/Status
//     Serial_COM Outputs/GVL_Serial_Com.stComOut_DREAM_CAT2_PTM_01/Ctrl <-> COM Outputs/Ctrl
//     Serial_COM Outputs/GVL_Serial_Com.stComOut_DREAM_CAT2_PTM_01/D[0] <-> COM Outputs/Data Out 0
//     Serial_COM Outputs/GVL_Serial_Com.stComOut_DREAM_CAT2_PTM_01/D[10] <-> COM Outputs/Data Out 10
//     Serial_COM Outputs/GVL_Serial_Com.stComOut_DREAM_CAT2_PTM_01/D[11] <-> COM Outputs/Data Out 11
//     Serial_COM Outputs/GVL_Serial_Com.stComOut_DREAM_CAT2_PTM_01/D[12] <-> COM Outputs/Data Out 12
//     Serial_COM Outputs/GVL_Serial_Com.stComOut_DREAM_CAT2_PTM_01/D[13] <-> COM Outputs/Data Out 13
//     Serial_COM Outputs/GVL_Serial_Com.stComOut_DREAM_CAT2_PTM_01/D[14] <-> COM Outputs/Data Out 14
//     Serial_COM Outputs/GVL_Serial_Com.stComOut_DREAM_CAT2_PTM_01/D[15] <-> COM Outputs/Data Out 15
//     Serial_COM Outputs/GVL_Serial_Com.stComOut_DREAM_CAT2_PTM_01/D[16] <-> COM Outputs/Data Out 16
//     Serial_COM Outputs/GVL_Serial_Com.stComOut_DREAM_CAT2_PTM_01/D[17] <-> COM Outputs/Data Out 17
//     Serial_COM Outputs/GVL_Serial_Com.stComOut_DREAM_CAT2_PTM_01/D[18] <-> COM Outputs/Data Out 18
//     Serial_COM Outputs/GVL_Serial_Com.stComOut_DREAM_CAT2_PTM_01/D[19] <-> COM Outputs/Data Out 19
//     Serial_COM Outputs/GVL_Serial_Com.stComOut_DREAM_CAT2_PTM_01/D[1] <-> COM Outputs/Data Out 1
//     Serial_COM Outputs/GVL_Serial_Com.stComOut_DREAM_CAT2_PTM_01/D[20] <-> COM Outputs/Data Out 20
//     Serial_COM Outputs/GVL_Serial_Com.stComOut_DREAM_CAT2_PTM_01/D[21] <-> COM Outputs/Data Out 21
//     Serial_COM Outputs/GVL_Serial_Com.stComOut_DREAM_CAT2_PTM_01/D[2] <-> COM Outputs/Data Out 2
//     Serial_COM Outputs/GVL_Serial_Com.stComOut_DREAM_CAT2_PTM_01/D[3] <-> COM Outputs/Data Out 3
//     Serial_COM Outputs/GVL_Serial_Com.stComOut_DREAM_CAT2_PTM_01/D[4] <-> COM Outputs/Data Out 4
//     Serial_COM Outputs/GVL_Serial_Com.stComOut_DREAM_CAT2_PTM_01/D[5] <-> COM Outputs/Data Out 5
//     Serial_COM Outputs/GVL_Serial_Com.stComOut_DREAM_CAT2_PTM_01/D[6] <-> COM Outputs/Data Out 6
//     Serial_COM Outputs/GVL_Serial_Com.stComOut_DREAM_CAT2_PTM_01/D[7] <-> COM Outputs/Data Out 7
//     Serial_COM Outputs/GVL_Serial_Com.stComOut_DREAM_CAT2_PTM_01/D[8] <-> COM Outputs/Data Out 8
//     Serial_COM Outputs/GVL_Serial_Com.stComOut_DREAM_CAT2_PTM_01/D[9] <-> COM Outputs/Data Out 9
//   lcls_plc_dream_vac Instance <-> Device 1 (EtherCAT)/R20_DRL_03_CX0_EK1200/R20_DRL_03_E15_EL1122/K4S8_DRL_04_EK0_EK1100/K4S8_DRL_04_E9_EL1004
//     PlcTask Inputs/GVL_VAC_VALVES.DREAM_ROUGH1_VRC_01.i_xClsLS <-> Channel 2/Input
//     PlcTask Inputs/GVL_VAC_VALVES.DREAM_ROUGH2_VRC_01.i_xClsLS <-> Channel 4/Input
//     PlcTask Inputs/GVL_VAC_VALVES.DREAM_ROUGH1_VRC_01.i_xOpnLS <-> Channel 1/Input
//     PlcTask Inputs/GVL_VAC_VALVES.DREAM_ROUGH2_VRC_01.i_xOpnLS <-> Channel 3/Input
//   lcls_plc_dream_vac Instance <-> Device 1 (EtherCAT)/R20_DRL_03_CX0_EK1200/R20_DRL_03_E15_EL1122/K4S8_DRL_04_EP1_EP4374-0002
//     PlcTask Inputs/GVL_VAC_GAUGES.DREAM_ROUGH1_GPI_02.i_iPRESS_R <-> AI Inputs Channel 1/Value
//     PlcTask Inputs/GVL_VAC_GAUGES.DREAM_ROUGH2_GPI_02.i_iPRESS_R <-> AI Inputs Channel 2/Value
//     PlcTask Outputs/GVL_VAC_VALVES.DREAM_ROUGH1_VFV_02.q_iRawPosition <-> AO Outputs Channel 3/Analog output
//     PlcTask Outputs/GVL_VAC_VALVES.DREAM_ROUGH2_VFV_02.q_iRawPosition <-> AO Outputs Channel 4/Analog output
//   lcls_plc_dream_vac Instance <-> Device 1 (EtherCAT)/R20_DRL_03_CX0_EK1200/R20_DRL_03_E15_EL1122/K4S8_DRL_04_EP2_EP4374-0002
//     PlcTask Inputs/GVL_VAC_GAUGES.DREAM_ROUGH2_GPI_03.i_iPRESS_R <-> AI Inputs Channel 1/Value
//     PlcTask Outputs/GVL_VAC_VALVES.DREAM_ROUGH2_VFV_03.q_iRawPosition <-> AO Outputs Channel 3/Analog output
//   lcls_plc_dream_vac Instance <-> Device 1 (EtherCAT)/R20_DRL_03_CX0_EK1200/R20_DRL_03_E15_EL1122/R03_DRL_01_EK1100/R03_DRL_01_E1_EL1004
//     PlcTask Inputs/GVL_VAC_GAUGES.DREAM_MC_GHC.i_xCH2_SEL <-> Channel 2/Input
//     PlcTask Inputs/GVL_VAC_GAUGES.DREAM_MC_GHC.i_xERR_CH1 <-> Channel 3/Input
//     PlcTask Inputs/GVL_VAC_GAUGES.DREAM_MC_GHC.i_xERR_CH2 <-> Channel 4/Input
//     PlcTask Inputs/GVL_VAC_GAUGES.DREAM_MC_GHC.i_xHV_ON <-> Channel 1/Input
//   lcls_plc_dream_vac Instance <-> Device 1 (EtherCAT)/R20_DRL_03_CX0_EK1200/R20_DRL_03_E15_EL1122/R03_DRL_01_EK1100/R03_DRL_01_E2_EL2624
//     PlcTask Outputs/GVL_VAC_GAUGES.DREAM_MC_GHC.q_xHV_DIS_CH1 <-> Channel 1/Output
//     PlcTask Outputs/GVL_VAC_GAUGES.DREAM_MC_GHC.q_xHV_DIS_CH2 <-> Channel 2/Output
//   lcls_plc_dream_vac Instance <-> Device 1 (EtherCAT)/R20_DRL_03_CX0_EK1200/R20_DRL_03_E15_EL1122/R03_DRL_01_EK1100/R03_DRL_01_E3_EL3174-0002
//     PlcTask Inputs/GVL_VAC_GAUGES.DREAM_MC_GHC.i_iPRESS_R_CH1 <-> AI Standard Channel 1/Value
//     PlcTask Inputs/GVL_VAC_GAUGES.DREAM_MC_GHC.i_iPRESS_R_CH2 <-> AI Standard Channel 2/Value
//   lcls_plc_dream_vac Instance <-> Device 1 (EtherCAT)/R20_DRL_03_CX0_EK1200/R20_DRL_03_E15_EL1122/WALL_E_PPL_01_EP1_EP4374-0002
//     PlcTask Inputs/GVL_VAC_GAUGES.DREAM_ROUGH1_GPI_01.i_iPRESS_R <-> AI Inputs Channel 1/Value
//     PlcTask Inputs/GVL_VAC_GAUGES.DREAM_ROUGH2_GPI_01.i_iPRESS_R <-> AI Inputs Channel 2/Value
//     PlcTask Outputs/GVL_VAC_VALVES.DREAM_ROUGH1_VFV_01.q_iRawPosition <-> AO Outputs Channel 3/Analog output
//     PlcTask Outputs/GVL_VAC_VALVES.DREAM_ROUGH2_VFV_01.q_iRawPosition <-> AO Outputs Channel 4/Analog output
//   lcls_plc_dream_vac Instance <-> Device 1 (EtherCAT)/R20_DRL_03_CX0_EK1200/R20_DRL_03_E4_EL1004
//     PlcTask Inputs/GVL_VAC_PUMPS.DREAM_DP2_PTM_01.i_xAtSpd <-> Channel 2/Input
//     PlcTask Inputs/GVL_VAC_PUMPS.DREAM_DP3_PTM_01.i_xAtSpd <-> Channel 4/Input
//     PlcTask Inputs/GVL_VAC_PUMPS.DREAM_DP2_PTM_01.i_xFaultNC <-> Channel 1/Input
//     PlcTask Inputs/GVL_VAC_PUMPS.DREAM_DP3_PTM_01.i_xFaultNC <-> Channel 3/Input
//   lcls_plc_dream_vac Instance <-> Device 1 (EtherCAT)/R20_DRL_03_CX0_EK1200/R20_DRL_03_E5_EL1004
//     PlcTask Inputs/GVL_VAC_PUMPS.DREAM_MC_PTM_01.i_xAtSpd <-> Channel 2/Input
//     PlcTask Inputs/GVL_VAC_PUMPS.DREAM_MC_PTM_02.i_xAtSpd <-> Channel 4/Input
//     PlcTask Inputs/GVL_VAC_PUMPS.DREAM_MC_PTM_01.i_xFaultNC <-> Channel 1/Input
//     PlcTask Inputs/GVL_VAC_PUMPS.DREAM_MC_PTM_02.i_xFaultNC <-> Channel 3/Input
//   lcls_plc_dream_vac Instance <-> Device 1 (EtherCAT)/R20_DRL_03_CX0_EK1200/R20_DRL_03_E7_EL2794
//     PlcTask Outputs/GVL_VAC_PUMPS.DREAM_DP2_PTM_01.q_RunDO <-> Channel 1/Output
//     PlcTask Outputs/GVL_VAC_PUMPS.DREAM_DP3_PTM_01.q_RunDO <-> Channel 3/Output
//     PlcTask Outputs/GVL_VAC_PUMPS.DREAM_MC_PTM_01.q_RunDO <-> Channel 2/Output
//     PlcTask Outputs/GVL_VAC_PUMPS.DREAM_MC_PTM_02.q_RunDO <-> Channel 4/Output
//   lcls_plc_dream_vac Instance <-> Device 1 (EtherCAT)/R20_DRL_03_CX0_EK1200/R20_DRL_03_E9_EL6001
//     Serial_COM Inputs/GVL_Serial_Com.stComIn_DREAM_DP2_PTM_01/D[0] <-> COM Inputs/Data In 0
//     Serial_COM Inputs/GVL_Serial_Com.stComIn_DREAM_DP2_PTM_01/D[10] <-> COM Inputs/Data In 10
//     Serial_COM Inputs/GVL_Serial_Com.stComIn_DREAM_DP2_PTM_01/D[11] <-> COM Inputs/Data In 11
//     Serial_COM Inputs/GVL_Serial_Com.stComIn_DREAM_DP2_PTM_01/D[12] <-> COM Inputs/Data In 12
//     Serial_COM Inputs/GVL_Serial_Com.stComIn_DREAM_DP2_PTM_01/D[13] <-> COM Inputs/Data In 13
//     Serial_COM Inputs/GVL_Serial_Com.stComIn_DREAM_DP2_PTM_01/D[14] <-> COM Inputs/Data In 14
//     Serial_COM Inputs/GVL_Serial_Com.stComIn_DREAM_DP2_PTM_01/D[15] <-> COM Inputs/Data In 15
//     Serial_COM Inputs/GVL_Serial_Com.stComIn_DREAM_DP2_PTM_01/D[16] <-> COM Inputs/Data In 16
//     Serial_COM Inputs/GVL_Serial_Com.stComIn_DREAM_DP2_PTM_01/D[17] <-> COM Inputs/Data In 17
//     Serial_COM Inputs/GVL_Serial_Com.stComIn_DREAM_DP2_PTM_01/D[18] <-> COM Inputs/Data In 18
//     Serial_COM Inputs/GVL_Serial_Com.stComIn_DREAM_DP2_PTM_01/D[19] <-> COM Inputs/Data In 19
//     Serial_COM Inputs/GVL_Serial_Com.stComIn_DREAM_DP2_PTM_01/D[1] <-> COM Inputs/Data In 1
//     Serial_COM Inputs/GVL_Serial_Com.stComIn_DREAM_DP2_PTM_01/D[20] <-> COM Inputs/Data In 20
//     Serial_COM Inputs/GVL_Serial_Com.stComIn_DREAM_DP2_PTM_01/D[21] <-> COM Inputs/Data In 21
//     Serial_COM Inputs/GVL_Serial_Com.stComIn_DREAM_DP2_PTM_01/D[2] <-> COM Inputs/Data In 2
//     Serial_COM Inputs/GVL_Serial_Com.stComIn_DREAM_DP2_PTM_01/D[3] <-> COM Inputs/Data In 3
//     Serial_COM Inputs/GVL_Serial_Com.stComIn_DREAM_DP2_PTM_01/D[4] <-> COM Inputs/Data In 4
//     Serial_COM Inputs/GVL_Serial_Com.stComIn_DREAM_DP2_PTM_01/D[5] <-> COM Inputs/Data In 5
//     Serial_COM Inputs/GVL_Serial_Com.stComIn_DREAM_DP2_PTM_01/D[6] <-> COM Inputs/Data In 6
//     Serial_COM Inputs/GVL_Serial_Com.stComIn_DREAM_DP2_PTM_01/D[7] <-> COM Inputs/Data In 7
//     Serial_COM Inputs/GVL_Serial_Com.stComIn_DREAM_DP2_PTM_01/D[8] <-> COM Inputs/Data In 8
//     Serial_COM Inputs/GVL_Serial_Com.stComIn_DREAM_DP2_PTM_01/D[9] <-> COM Inputs/Data In 9
//     Serial_COM Inputs/GVL_Serial_Com.stComIn_DREAM_DP2_PTM_01/Status <-> COM Inputs/Status
//     Serial_COM Outputs/GVL_Serial_Com.stComOut_DREAM_DP2_PTM_01/Ctrl <-> COM Outputs/Ctrl
//     Serial_COM Outputs/GVL_Serial_Com.stComOut_DREAM_DP2_PTM_01/D[0] <-> COM Outputs/Data Out 0
//     Serial_COM Outputs/GVL_Serial_Com.stComOut_DREAM_DP2_PTM_01/D[10] <-> COM Outputs/Data Out 10
//     Serial_COM Outputs/GVL_Serial_Com.stComOut_DREAM_DP2_PTM_01/D[11] <-> COM Outputs/Data Out 11
//     Serial_COM Outputs/GVL_Serial_Com.stComOut_DREAM_DP2_PTM_01/D[12] <-> COM Outputs/Data Out 12
//     Serial_COM Outputs/GVL_Serial_Com.stComOut_DREAM_DP2_PTM_01/D[13] <-> COM Outputs/Data Out 13
//     Serial_COM Outputs/GVL_Serial_Com.stComOut_DREAM_DP2_PTM_01/D[14] <-> COM Outputs/Data Out 14
//     Serial_COM Outputs/GVL_Serial_Com.stComOut_DREAM_DP2_PTM_01/D[15] <-> COM Outputs/Data Out 15
//     Serial_COM Outputs/GVL_Serial_Com.stComOut_DREAM_DP2_PTM_01/D[16] <-> COM Outputs/Data Out 16
//     Serial_COM Outputs/GVL_Serial_Com.stComOut_DREAM_DP2_PTM_01/D[17] <-> COM Outputs/Data Out 17
//     Serial_COM Outputs/GVL_Serial_Com.stComOut_DREAM_DP2_PTM_01/D[18] <-> COM Outputs/Data Out 18
//     Serial_COM Outputs/GVL_Serial_Com.stComOut_DREAM_DP2_PTM_01/D[19] <-> COM Outputs/Data Out 19
//     Serial_COM Outputs/GVL_Serial_Com.stComOut_DREAM_DP2_PTM_01/D[1] <-> COM Outputs/Data Out 1
//     Serial_COM Outputs/GVL_Serial_Com.stComOut_DREAM_DP2_PTM_01/D[20] <-> COM Outputs/Data Out 20
//     Serial_COM Outputs/GVL_Serial_Com.stComOut_DREAM_DP2_PTM_01/D[21] <-> COM Outputs/Data Out 21
//     Serial_COM Outputs/GVL_Serial_Com.stComOut_DREAM_DP2_PTM_01/D[2] <-> COM Outputs/Data Out 2
//     Serial_COM Outputs/GVL_Serial_Com.stComOut_DREAM_DP2_PTM_01/D[3] <-> COM Outputs/Data Out 3
//     Serial_COM Outputs/GVL_Serial_Com.stComOut_DREAM_DP2_PTM_01/D[4] <-> COM Outputs/Data Out 4
//     Serial_COM Outputs/GVL_Serial_Com.stComOut_DREAM_DP2_PTM_01/D[5] <-> COM Outputs/Data Out 5
//     Serial_COM Outputs/GVL_Serial_Com.stComOut_DREAM_DP2_PTM_01/D[6] <-> COM Outputs/Data Out 6
//     Serial_COM Outputs/GVL_Serial_Com.stComOut_DREAM_DP2_PTM_01/D[7] <-> COM Outputs/Data Out 7
//     Serial_COM Outputs/GVL_Serial_Com.stComOut_DREAM_DP2_PTM_01/D[8] <-> COM Outputs/Data Out 8
//     Serial_COM Outputs/GVL_Serial_Com.stComOut_DREAM_DP2_PTM_01/D[9] <-> COM Outputs/Data Out 9

// ---- POUs/TD400_Test/FB_OERLIKON_TD400_COM.TcPOU
FUNCTION_BLOCK FB_OERLIKON_TD400_COM
VAR_INPUT
END_VAR
VAR
    tTimeOut : TIME := TIME#1S0MS;
    fbTD400SerialDriver : FB_TD400SerialDriver;
END_VAR
VAR_IN_OUT
    SerialRXBuffer : ComBuffer;
    SerialTXBuffer : ComBuffer;
    stTD400Control : ST_TD400Control;
END_VAR
VAR_OUTPUT
    stTD400Status : ST_TD400Status;
END_VAR

(* This program is called from Serial PTM IO *)

(* scan the pumps one at a time *)//MG???
fbTD400SerialDriver(
    i_xExecute:= TRUE,
    i_tTimeOut:= tTimeOut,
    i_wControlWord:= 16#0000,
    iq_stControl:= stTD400Control,
    iq_stSerialRXBuffer:= SerialRXBuffer,
    iq_stSerialTXBuffer:= SerialTXBuffer,
    q_xDone=> ,
    q_xError=> ,
    q_xTimeout=> ,
    q_sResult=> ,
    q_stStatus=> stTD400Status);

IF fbTD400SerialDriver.q_xDone
   OR fbTD400SerialDriver.q_xError
   OR fbTD400SerialDriver.q_xTimeout THEN
         (* reset for next time *)
        fbTD400SerialDriver(i_xExecute:= FALSE, iq_stSerialRXBuffer:= SerialRXBuffer, iq_stSerialTXBuffer:= SerialTXBuffer, iq_stControl:= stTD400Control);
END_IF

END_FUNCTION_BLOCK

// ---- POUs/TD400_Test/FB_OERLIKON_TD400_TO_PTM.TcPOU
FUNCTION_BLOCK FB_OERLIKON_TD400_TO_PTM
VAR_IN_OUT
    iq_stPTM : ST_LeyboldPTM;
    iq_stTD400Status : ST_TD400Status;
    iq_stTD400Control : ST_TD400Control;
END_VAR
VAR
END_VAR

(* This function block is used to map the IO points from the Oerlikon TD400 structures
to the generic turbo structures *)
//Use this function to map IO as a temporary solution if we don't change method FB_PTM_TurboDrive.M_Serial_IO and ST_LeyboldPTM structure

(* Readbacks *)
iq_stPTM.i_xAccel := iq_stTD400Status.wStatusWord.4;
iq_stPTM.i_xDecel := iq_stTD400Status.wStatusWord.5;
//iq_stPTM.i_xAtSpd := iq_stTD400Status.wStatusWord.10;
iq_stPTM.q_xRemote := iq_stTD400Status.wStatusWord.15; (* Remote control enabled *)
iq_stPTM.i_diCurSpd := WORD_TO_DINT(iq_stTD400Status.wFrequency_P3);
iq_stPTM.i_rCurrentMon := WORD_TO_INT(iq_stTD400Status.wMotorCurrent_P5)*0.1; (*Current in units 0.1 A, TD400 Interface manual page 6*)
iq_stPTM.i_diPwr := REAL_TO_DINT(WORD_TO_DINT(iq_stTD400Status.wMotorCurrent_P5 * iq_stTD400Status.wVoltage_P4)*0.1); (*Current in units 0.1 A, TD400 Interface manual page 6*)
iq_stPTM.i_diElecTemp := WORD_TO_DINT(iq_stTD400Status.wConverterTemp_P11);
iq_stPTM.i_rTempMon := WORD_TO_INT(iq_stTD400Status.wPumpTemp_P127);

(* Faults and warnings *)
//iq_stPTM.xFault := iq_stTD400Status.wStatusWord.3;
iq_stPTM.i_xTempFault := iq_stTD400Status.wStatusWord.7; (* specified as a temperature warning but it could be a fault *)
iq_stPTM.i_xWarn := iq_stTD400Status.wStatusWord.14; (* warning summary bit *)

(* Controls *)
iq_stTD400Control.wSetSetpointFreq_P24 := LIMIT (iq_stTD400Status.wMinSetpointFreq_P19, iq_stTD400Control.wSetSetpointFreq_P24, iq_stTD400Status.wMaxSetpointFreq_P18);

END_FUNCTION_BLOCK
